DATA_BLOCK "DB_MFC_ErrorCode"
{ S7_Optimized_Access := 'TRUE' }
VERSION : 0.1
NON_RETAIN
   VAR
      PEC { ExternalAccessible := 'False'; ExternalVisible := 'False'; ExternalWritable := 'False'} : Struct
         Jam { ExternalAccessible := 'False'; ExternalVisible := 'False'; ExternalWritable := 'False'} : Int;
      END_STRUCT;
      PECUpdate { ExternalAccessible := 'False'; ExternalVisible := 'False'; ExternalWritable := 'False'} : Struct
         TooManyLost { ExternalAccessible := 'False'; ExternalVisible := 'False'; ExternalWritable := 'False'} : Int;
         LowPerformance { ExternalAccessible := 'False'; ExternalVisible := 'False'; ExternalWritable := 'False'} : Int;
         Jam { ExternalAccessible := 'False'; ExternalVisible := 'False'; ExternalWritable := 'False'} : Int;
      END_STRUCT;
      VFD { ExternalAccessible := 'False'; ExternalVisible := 'False'; ExternalWritable := 'False'} : Struct
         PNSlaveNotonline { ExternalAccessible := 'False'; ExternalVisible := 'False'; ExternalWritable := 'False'} : Int;
         PNSlaveError { ExternalAccessible := 'False'; ExternalVisible := 'False'; ExternalWritable := 'False'} : Int;
         InternalError { ExternalAccessible := 'False'; ExternalVisible := 'False'; ExternalWritable := 'False'} : Int;
         InternalWarning { ExternalAccessible := 'False'; ExternalVisible := 'False'; ExternalWritable := 'False'} : Int;
         CommunicationErrorMovikit { ExternalAccessible := 'False'; ExternalVisible := 'False'; ExternalWritable := 'False'} : Int;
         VFDRunningFeedbackError { ExternalAccessible := 'False'; ExternalVisible := 'False'; ExternalWritable := 'False'} : Int;
         PNSlaveWarning { ExternalAccessible := 'False'; ExternalVisible := 'False'; ExternalWritable := 'False'} : Int;
      END_STRUCT;
      Conveyor { ExternalAccessible := 'False'; ExternalVisible := 'False'; ExternalWritable := 'False'} : Struct
         ErrorCode { ExternalAccessible := 'False'; ExternalVisible := 'False'; ExternalWritable := 'False'} : Int;
         SubErrorCode { ExternalAccessible := 'False'; ExternalVisible := 'False'; ExternalWritable := 'False'} : Int;
         PNSlaveNotonline { ExternalAccessible := 'False'; ExternalVisible := 'False'; ExternalWritable := 'False'} : Int;
         PNSlaveError { ExternalAccessible := 'False'; ExternalVisible := 'False'; ExternalWritable := 'False'} : Int;
         InternalError { ExternalAccessible := 'False'; ExternalVisible := 'False'; ExternalWritable := 'False'} : Int;
         InternalWarning { ExternalAccessible := 'False'; ExternalVisible := 'False'; ExternalWritable := 'False'} : Int;
         CommunicationErrorMovikit { ExternalAccessible := 'False'; ExternalVisible := 'False'; ExternalWritable := 'False'} : Int;
         VFDRunningFeedbackError { ExternalAccessible := 'False'; ExternalVisible := 'False'; ExternalWritable := 'False'} : Int;
         PNSlaveWarning { ExternalAccessible := 'False'; ExternalVisible := 'False'; ExternalWritable := 'False'} : Int;
      END_STRUCT;
      Caljan { ExternalAccessible := 'False'; ExternalVisible := 'False'; ExternalWritable := 'False'} : Struct
         PNSlaveNotOnline { ExternalAccessible := 'False'; ExternalVisible := 'False'; ExternalWritable := 'False'} : Int;
         PNSlaveError { ExternalAccessible := 'False'; ExternalVisible := 'False'; ExternalWritable := 'False'} : Int;
         PNSlaveWarning { ExternalAccessible := 'False'; ExternalVisible := 'False'; ExternalWritable := 'False'} : Int;
         Disabled { ExternalAccessible := 'False'; ExternalVisible := 'False'; ExternalWritable := 'False'} : Int;
         VFDError { ExternalAccessible := 'False'; ExternalVisible := 'False'; ExternalWritable := 'False'} : Int;
         NotHealthy { ExternalAccessible := 'False'; ExternalVisible := 'False'; ExternalWritable := 'False'} : Int;
         StoreMode { ExternalAccessible := 'False'; ExternalVisible := 'False'; ExternalWritable := 'False'} : Int;
         RunMode { ExternalAccessible := 'False'; ExternalVisible := 'False'; ExternalWritable := 'False'} : Int;
         ChuteBlocked { ExternalAccessible := 'False'; ExternalVisible := 'False'; ExternalWritable := 'False'} : Int;
         Jam { ExternalAccessible := 'False'; ExternalVisible := 'False'; ExternalWritable := 'False'} : Int;
      END_STRUCT;
      ArmDiverter { ExternalAccessible := 'False'; ExternalVisible := 'False'; ExternalWritable := 'False'} : Struct
         TimeoutError { ExternalAccessible := 'False'; ExternalVisible := 'False'; ExternalWritable := 'False'} : Int;
         LimitHomeError { ExternalAccessible := 'False'; ExternalVisible := 'False'; ExternalWritable := 'False'} : Int;
         LimitDivertError { ExternalAccessible := 'False'; ExternalVisible := 'False'; ExternalWritable := 'False'} : Int;
         PXHomeError { ExternalAccessible := 'False'; ExternalVisible := 'False'; ExternalWritable := 'False'} : Int;
         PXDivertError { ExternalAccessible := 'False'; ExternalVisible := 'False'; ExternalWritable := 'False'} : Int;
         AtHomePosition { ExternalAccessible := 'False'; ExternalVisible := 'False'; ExternalWritable := 'False'} : Int;
         AtDivertPosition { ExternalAccessible := 'False'; ExternalVisible := 'False'; ExternalWritable := 'False'} : Int;
         ReferencError { ExternalAccessible := 'False'; ExternalVisible := 'False'; ExternalWritable := 'False'} : Int;
         ParcelDivertError { ExternalAccessible := 'False'; ExternalVisible := 'False'; ExternalWritable := 'False'} : Int;
      END_STRUCT;
      MCP { ExternalAccessible := 'False'; ExternalVisible := 'False'; ExternalWritable := 'False'} : Struct
         PN_PN_MSP_PNSlaveNotOnline { ExternalAccessible := 'False'; ExternalVisible := 'False'; ExternalWritable := 'False'} : Int;   // PNPN coupler is not online
         PN_PN_MSP_PNSlaveError { ExternalAccessible := 'False'; ExternalVisible := 'False'; ExternalWritable := 'False'} : Int;   // PNPN coupler has an error
         PN_PN_MSP_PNSlaveWarning { ExternalAccessible := 'False'; ExternalVisible := 'False'; ExternalWritable := 'False'} : Int;   // PNPN coupler has a warning
         IOModule_PNSlaveNotOnline { ExternalAccessible := 'False'; ExternalVisible := 'False'; ExternalWritable := 'False'} : Int;   // I/O Module is not online
         IOModule_PNSlaveError { ExternalAccessible := 'False'; ExternalVisible := 'False'; ExternalWritable := 'False'} : Int;   // I/O Module has an error
         IOModule_PNSlaveWarning { ExternalAccessible := 'False'; ExternalVisible := 'False'; ExternalWritable := 'False'} : Int;   // I/O Module has a warning
         ScalanceSwitchPNSlaveNotOnline { ExternalAccessible := 'False'; ExternalVisible := 'False'; ExternalWritable := 'False'} : Int;   // Scalance switch is not online (Switch 1)
         ScalanceSwitchPNSlaveError { ExternalAccessible := 'False'; ExternalVisible := 'False'; ExternalWritable := 'False'} : Int;   // Scalance switch has an error (Switch 1)
         ScalanceSwitchPNSlaveWarning { ExternalAccessible := 'False'; ExternalVisible := 'False'; ExternalWritable := 'False'} : Int;   // Scalance switch has a warning (Switch 1)
         "2ndScalanceSwitchPNSlaveNotOnline" { ExternalAccessible := 'False'; ExternalVisible := 'False'; ExternalWritable := 'False'} : Int;   // Scalance switch is not online (Switch 2)
         "2ndScalanceSwitchPNSlaveError" { ExternalAccessible := 'False'; ExternalVisible := 'False'; ExternalWritable := 'False'} : Int;   // Scalance switch has an error (Switch 2)
         "2ndScalanceSwitchPNSlaveWarning" { ExternalAccessible := 'False'; ExternalVisible := 'False'; ExternalWritable := 'False'} : Int;   // Scalance switch has a warning (Switch 2)
         Singulator_PNSlaveNotOnline { ExternalAccessible := 'False'; ExternalVisible := 'False'; ExternalWritable := 'False'} : Int;   // Singulator coupler is not online
         Singulator_PNSlaveError { ExternalAccessible := 'False'; ExternalVisible := 'False'; ExternalWritable := 'False'} : Int;   // Singulator coupler has an error
         Singulator_PNSlaveWarning { ExternalAccessible := 'False'; ExternalVisible := 'False'; ExternalWritable := 'False'} : Int;   // Singulator coupler has a warning
         IPS_PNSlaveNotOnline { ExternalAccessible := 'False'; ExternalVisible := 'False'; ExternalWritable := 'False'} : Int;   // IPS is not online
         IPS_PNSlaveError { ExternalAccessible := 'False'; ExternalVisible := 'False'; ExternalWritable := 'False'} : Int;   // IPS has an error
         IPS_PNSlaveWarning { ExternalAccessible := 'False'; ExternalVisible := 'False'; ExternalWritable := 'False'} : Int;   // IPS has a warning
         UPSSwitchTripped { ExternalAccessible := 'False'; ExternalVisible := 'False'; ExternalWritable := 'False'} : Int;   // Unit Power Supply switch tripped
         FireAlarmActive { ExternalAccessible := 'False'; ExternalVisible := 'False'; ExternalWritable := 'False'} : Int;   // Fire alarm active when the signal is true
         PS_201T1_Tripped { ExternalAccessible := 'False'; ExternalVisible := 'False'; ExternalWritable := 'False'} : Int;   // TRUE if power supply 201T1 tripped
         "230VAC_CB101F4Tripped" { ExternalAccessible := 'False'; ExternalVisible := 'False'; ExternalWritable := 'False'} : Int;   // TRUE if MCP circuit breaker 101F4 tripped
         "230VAC_CB102F1Tripped" { ExternalAccessible := 'False'; ExternalVisible := 'False'; ExternalWritable := 'False'} : Int;   // TRUE if MCP circuit breaker 102F1 tripped
         "24VDC_CB201F1Tripped" { ExternalAccessible := 'False'; ExternalVisible := 'False'; ExternalWritable := 'False'} : Int;   // TRUE if MCP circuit breaker 201F1 tripped
         "24VDC_CB205F5Tripped" { ExternalAccessible := 'False'; ExternalVisible := 'False'; ExternalWritable := 'False'} : Int;   // TRUE if MCP circuit breaker 205F5 tripped
         Spare_1 { ExternalAccessible := 'False'; ExternalVisible := 'False'; ExternalWritable := 'False'} : Int;   // Spare
         Spare_2 { ExternalAccessible := 'False'; ExternalVisible := 'False'; ExternalWritable := 'False'} : Int;   // Spare
         Spare_3 { ExternalAccessible := 'False'; ExternalVisible := 'False'; ExternalWritable := 'False'} : Int;   // Spare
         RackSlotError { ExternalAccessible := 'False'; ExternalVisible := 'False'; ExternalWritable := 'False'} : Array[0..31] of Int;   // One of the main rack slots has an error
         IOModuleSlotError { ExternalAccessible := 'False'; ExternalVisible := 'False'; ExternalWritable := 'False'} : Array[0..31] of Int;   // Module error
      END_STRUCT;
      RIO { ExternalAccessible := 'False'; ExternalVisible := 'False'; ExternalWritable := 'False'} : Struct
         PNSlaveNotOnline { ExternalAccessible := 'False'; ExternalVisible := 'False'; ExternalWritable := 'False'} : Int;
         PNSlaveError { ExternalAccessible := 'False'; ExternalVisible := 'False'; ExternalWritable := 'False'} : Int;
         PNSlaveWarning { ExternalAccessible := 'False'; ExternalVisible := 'False'; ExternalWritable := 'False'} : Int;
         ET200sp_ErrorModule { ExternalAccessible := 'False'; ExternalVisible := 'False'; ExternalWritable := 'False'} : Array[0..31] of Int;
      END_STRUCT;
      Connect { ExternalAccessible := 'False'; ExternalVisible := 'False'; ExternalWritable := 'False'} : Struct
         CommunicationFault { ExternalAccessible := 'False'; ExternalVisible := 'False'; ExternalWritable := 'False'} : Int;
      END_STRUCT;
      ConveyorInterface { ExternalAccessible := 'False'; ExternalVisible := 'False'; ExternalWritable := 'False'} : Struct
         InternalErrorTracking { ExternalAccessible := 'False'; ExternalVisible := 'False'; ExternalWritable := 'False'} : Int;
         InternalWarningTracking { ExternalAccessible := 'False'; ExternalVisible := 'False'; ExternalWritable := 'False'} : Int;
         Disconnected { ExternalAccessible := 'False'; ExternalVisible := 'False'; ExternalWritable := 'False'} : Int;
      END_STRUCT;
      PDP { ExternalAccessible := 'False'; ExternalVisible := 'False'; ExternalWritable := 'False'} : Struct
         CircuitBreakersTripped { ExternalAccessible := 'False'; ExternalVisible := 'False'; ExternalWritable := 'False'} : Int;
         CircuitBreakerStateF100_F200_F300 { ExternalAccessible := 'False'; ExternalVisible := 'False'; ExternalWritable := 'False'} : Int;
         CircuitBreakerStatePM { ExternalAccessible := 'False'; ExternalVisible := 'False'; ExternalWritable := 'False'} : Int;
         CircuitBreakerTrippedF101 { ExternalAccessible := 'False'; ExternalVisible := 'False'; ExternalWritable := 'False'} : Int;
         CircuitBreakerTrippedF102 { ExternalAccessible := 'False'; ExternalVisible := 'False'; ExternalWritable := 'False'} : Int;
         CircuitBreakerTrippedF103 { ExternalAccessible := 'False'; ExternalVisible := 'False'; ExternalWritable := 'False'} : Int;
         CircuitBreakerTrippedF104 { ExternalAccessible := 'False'; ExternalVisible := 'False'; ExternalWritable := 'False'} : Int;
         CircuitBreakerTrippedF105 { ExternalAccessible := 'False'; ExternalVisible := 'False'; ExternalWritable := 'False'} : Int;
         CircuitBreakerTrippedF106 { ExternalAccessible := 'False'; ExternalVisible := 'False'; ExternalWritable := 'False'} : Int;
         CircuitBreakerTrippedF107 { ExternalAccessible := 'False'; ExternalVisible := 'False'; ExternalWritable := 'False'} : Int;
         CircuitBreakerTrippedF108 { ExternalAccessible := 'False'; ExternalVisible := 'False'; ExternalWritable := 'False'} : Int;
         CircuitBreakerTrippedF109 { ExternalAccessible := 'False'; ExternalVisible := 'False'; ExternalWritable := 'False'} : Int;
         CircuitBreakerTrippedF110 { ExternalAccessible := 'False'; ExternalVisible := 'False'; ExternalWritable := 'False'} : Int;
         CircuitBreakerTrippedF111 { ExternalAccessible := 'False'; ExternalVisible := 'False'; ExternalWritable := 'False'} : Int;
         CircuitBreakerTrippedF112 { ExternalAccessible := 'False'; ExternalVisible := 'False'; ExternalWritable := 'False'} : Int;
         CircuitBreakerTrippedF113 { ExternalAccessible := 'False'; ExternalVisible := 'False'; ExternalWritable := 'False'} : Int;
         CircuitBreakerTrippedF114 { ExternalAccessible := 'False'; ExternalVisible := 'False'; ExternalWritable := 'False'} : Int;
         CircuitBreakerTrippedF115 { ExternalAccessible := 'False'; ExternalVisible := 'False'; ExternalWritable := 'False'} : Int;
         CircuitBreakerTrippedF116 { ExternalAccessible := 'False'; ExternalVisible := 'False'; ExternalWritable := 'False'} : Int;
         CircuitBreakerTrippedF117 { ExternalAccessible := 'False'; ExternalVisible := 'False'; ExternalWritable := 'False'} : Int;
         CircuitBreakerTrippedF118 { ExternalAccessible := 'False'; ExternalVisible := 'False'; ExternalWritable := 'False'} : Int;
         CircuitBreakerTrippedF119 { ExternalAccessible := 'False'; ExternalVisible := 'False'; ExternalWritable := 'False'} : Int;
         CircuitBreakerTrippedF120 { ExternalAccessible := 'False'; ExternalVisible := 'False'; ExternalWritable := 'False'} : Int;
         CircuitBreakerTrippedF121 { ExternalAccessible := 'False'; ExternalVisible := 'False'; ExternalWritable := 'False'} : Int;
         CircuitBreakerTrippedF122 { ExternalAccessible := 'False'; ExternalVisible := 'False'; ExternalWritable := 'False'} : Int;
         CircuitBreakerTrippedF123 { ExternalAccessible := 'False'; ExternalVisible := 'False'; ExternalWritable := 'False'} : Int;
         CircuitBreakerTrippedF124 { ExternalAccessible := 'False'; ExternalVisible := 'False'; ExternalWritable := 'False'} : Int;
         CircuitBreakerTrippedF125 { ExternalAccessible := 'False'; ExternalVisible := 'False'; ExternalWritable := 'False'} : Int;
         CircuitBreakerTrippedF126 { ExternalAccessible := 'False'; ExternalVisible := 'False'; ExternalWritable := 'False'} : Int;
         CircuitBreakerTrippedF127 { ExternalAccessible := 'False'; ExternalVisible := 'False'; ExternalWritable := 'False'} : Int;
         CircuitBreakerTrippedF128 { ExternalAccessible := 'False'; ExternalVisible := 'False'; ExternalWritable := 'False'} : Int;
         CircuitBreakerTrippedF129 { ExternalAccessible := 'False'; ExternalVisible := 'False'; ExternalWritable := 'False'} : Int;
         CircuitBreakerTrippedF130 { ExternalAccessible := 'False'; ExternalVisible := 'False'; ExternalWritable := 'False'} : Int;
         CircuitBreakerTrippedF131 { ExternalAccessible := 'False'; ExternalVisible := 'False'; ExternalWritable := 'False'} : Int;
         CircuitBreakerTrippedF132 { ExternalAccessible := 'False'; ExternalVisible := 'False'; ExternalWritable := 'False'} : Int;
         CircuitBreakerTrippedF133 { ExternalAccessible := 'False'; ExternalVisible := 'False'; ExternalWritable := 'False'} : Int;
         CircuitBreakerTrippedF134 { ExternalAccessible := 'False'; ExternalVisible := 'False'; ExternalWritable := 'False'} : Int;
         CircuitBreakerTrippedF135 { ExternalAccessible := 'False'; ExternalVisible := 'False'; ExternalWritable := 'False'} : Int;
         CircuitBreakerTrippedF201 { ExternalAccessible := 'False'; ExternalVisible := 'False'; ExternalWritable := 'False'} : Int;
         CircuitBreakerTrippedF202 { ExternalAccessible := 'False'; ExternalVisible := 'False'; ExternalWritable := 'False'} : Int;
         CircuitBreakerTrippedF203 { ExternalAccessible := 'False'; ExternalVisible := 'False'; ExternalWritable := 'False'} : Int;
         CircuitBreakerTrippedF204 { ExternalAccessible := 'False'; ExternalVisible := 'False'; ExternalWritable := 'False'} : Int;
         CircuitBreakerTrippedF205 { ExternalAccessible := 'False'; ExternalVisible := 'False'; ExternalWritable := 'False'} : Int;
         CircuitBreakerTrippedF206 { ExternalAccessible := 'False'; ExternalVisible := 'False'; ExternalWritable := 'False'} : Int;
         CircuitBreakerTrippedF207 { ExternalAccessible := 'False'; ExternalVisible := 'False'; ExternalWritable := 'False'} : Int;
         CircuitBreakerTrippedF208 { ExternalAccessible := 'False'; ExternalVisible := 'False'; ExternalWritable := 'False'} : Int;
         CircuitBreakerTrippedF209 { ExternalAccessible := 'False'; ExternalVisible := 'False'; ExternalWritable := 'False'} : Int;
         CircuitBreakerTrippedF210 { ExternalAccessible := 'False'; ExternalVisible := 'False'; ExternalWritable := 'False'} : Int;
         CircuitBreakerTrippedF211 { ExternalAccessible := 'False'; ExternalVisible := 'False'; ExternalWritable := 'False'} : Int;
         CircuitBreakerTrippedF212 { ExternalAccessible := 'False'; ExternalVisible := 'False'; ExternalWritable := 'False'} : Int;
         CircuitBreakerTrippedF213 { ExternalAccessible := 'False'; ExternalVisible := 'False'; ExternalWritable := 'False'} : Int;
         CircuitBreakerTrippedF214 { ExternalAccessible := 'False'; ExternalVisible := 'False'; ExternalWritable := 'False'} : Int;
         CircuitBreakerTrippedF215 { ExternalAccessible := 'False'; ExternalVisible := 'False'; ExternalWritable := 'False'} : Int;
         CircuitBreakerTrippedF216 { ExternalAccessible := 'False'; ExternalVisible := 'False'; ExternalWritable := 'False'} : Int;
         CircuitBreakerTrippedF217 { ExternalAccessible := 'False'; ExternalVisible := 'False'; ExternalWritable := 'False'} : Int;
         CircuitBreakerTrippedF218 { ExternalAccessible := 'False'; ExternalVisible := 'False'; ExternalWritable := 'False'} : Int;
         CircuitBreakerTrippedF219 { ExternalAccessible := 'False'; ExternalVisible := 'False'; ExternalWritable := 'False'} : Int;
         CircuitBreakerTrippedF220 { ExternalAccessible := 'False'; ExternalVisible := 'False'; ExternalWritable := 'False'} : Int;
         CircuitBreakerTrippedF221 { ExternalAccessible := 'False'; ExternalVisible := 'False'; ExternalWritable := 'False'} : Int;
         CircuitBreakerTrippedF222 { ExternalAccessible := 'False'; ExternalVisible := 'False'; ExternalWritable := 'False'} : Int;
         CircuitBreakerTrippedF223 { ExternalAccessible := 'False'; ExternalVisible := 'False'; ExternalWritable := 'False'} : Int;
         CircuitBreakerTrippedF224 { ExternalAccessible := 'False'; ExternalVisible := 'False'; ExternalWritable := 'False'} : Int;
         CircuitBreakerTrippedF225 { ExternalAccessible := 'False'; ExternalVisible := 'False'; ExternalWritable := 'False'} : Int;
         CircuitBreakerTrippedF226 { ExternalAccessible := 'False'; ExternalVisible := 'False'; ExternalWritable := 'False'} : Int;
         CircuitBreakerTrippedF227 { ExternalAccessible := 'False'; ExternalVisible := 'False'; ExternalWritable := 'False'} : Int;
         CircuitBreakerTrippedF228 { ExternalAccessible := 'False'; ExternalVisible := 'False'; ExternalWritable := 'False'} : Int;
         CircuitBreakerTrippedF229 { ExternalAccessible := 'False'; ExternalVisible := 'False'; ExternalWritable := 'False'} : Int;
         CircuitBreakerTrippedF501 { ExternalAccessible := 'False'; ExternalVisible := 'False'; ExternalWritable := 'False'} : Int;
         CircuitBreakerTrippedF502 { ExternalAccessible := 'False'; ExternalVisible := 'False'; ExternalWritable := 'False'} : Int;
         CircuitBreakerTrippedF503 { ExternalAccessible := 'False'; ExternalVisible := 'False'; ExternalWritable := 'False'} : Int;
         CircuitBreakerTrippedF504 { ExternalAccessible := 'False'; ExternalVisible := 'False'; ExternalWritable := 'False'} : Int;
         CircuitBreakerTrippedF505 { ExternalAccessible := 'False'; ExternalVisible := 'False'; ExternalWritable := 'False'} : Int;
         CircuitBreakerTrippedF506 { ExternalAccessible := 'False'; ExternalVisible := 'False'; ExternalWritable := 'False'} : Int;
         CircuitBreakerTrippedF507 { ExternalAccessible := 'False'; ExternalVisible := 'False'; ExternalWritable := 'False'} : Int;
         CircuitBreakerTrippedF508 { ExternalAccessible := 'False'; ExternalVisible := 'False'; ExternalWritable := 'False'} : Int;
         CircuitBreakerTrippedF509 { ExternalAccessible := 'False'; ExternalVisible := 'False'; ExternalWritable := 'False'} : Int;
         CircuitBreakerTrippedF510 { ExternalAccessible := 'False'; ExternalVisible := 'False'; ExternalWritable := 'False'} : Int;
         CircuitBreakerTrippedF511 { ExternalAccessible := 'False'; ExternalVisible := 'False'; ExternalWritable := 'False'} : Int;
         CircuitBreakerTrippedF512 { ExternalAccessible := 'False'; ExternalVisible := 'False'; ExternalWritable := 'False'} : Int;
      END_STRUCT;
      TCPIPConnection { ExternalAccessible := 'False'; ExternalVisible := 'False'; ExternalWritable := 'False'} : Struct
         CommunicationFault { ExternalAccessible := 'False'; ExternalVisible := 'False'; ExternalWritable := 'False'} : Int;
      END_STRUCT;
      PNNode { ExternalAccessible := 'False'; ExternalVisible := 'False'; ExternalWritable := 'False'} : Struct
         PNSlaveNotOnline { ExternalAccessible := 'False'; ExternalVisible := 'False'; ExternalWritable := 'False'} : Int;
         PNSlaveError { ExternalAccessible := 'False'; ExternalVisible := 'False'; ExternalWritable := 'False'} : Int;
         PNSlaveWarning { ExternalAccessible := 'False'; ExternalVisible := 'False'; ExternalWritable := 'False'} : Int;
      END_STRUCT;
      EStop { ExternalAccessible := 'False'; ExternalVisible := 'False'; ExternalWritable := 'False'} : Struct
         EStop { ExternalAccessible := 'False'; ExternalVisible := 'False'; ExternalWritable := 'False'} : Int;
      END_STRUCT;
      Outfeed2States { ExternalAccessible := 'False'; ExternalVisible := 'False'; ExternalWritable := 'False'} : Struct
         ChuteFull { ExternalAccessible := 'False'; ExternalVisible := 'False'; ExternalWritable := 'False'} : Int;
         ChuteHalfFull { ExternalAccessible := 'False'; ExternalVisible := 'False'; ExternalWritable := 'False'} : Int;
         ChuteDisabled { ExternalAccessible := 'False'; ExternalVisible := 'False'; ExternalWritable := 'False'} : Int;
      END_STRUCT;
      Rapiscan { ExternalAccessible := 'False'; ExternalVisible := 'False'; ExternalWritable := 'False'} : Struct
         XrayEnergised { ExternalAccessible := 'False'; ExternalVisible := 'False'; ExternalWritable := 'False'} : Int;
         XrayFault { ExternalAccessible := 'False'; ExternalVisible := 'False'; ExternalWritable := 'False'} : Int;
         XrayRdyRCV { ExternalAccessible := 'False'; ExternalVisible := 'False'; ExternalWritable := 'False'} : Int;
         XrayRdySend { ExternalAccessible := 'False'; ExternalVisible := 'False'; ExternalWritable := 'False'} : Int;
         BagScanning { ExternalAccessible := 'False'; ExternalVisible := 'False'; ExternalWritable := 'False'} : Int;
         TransportMode { ExternalAccessible := 'False'; ExternalVisible := 'False'; ExternalWritable := 'False'} : Int;
         BackBelt { ExternalAccessible := 'False'; ExternalVisible := 'False'; ExternalWritable := 'False'} : Int;
      END_STRUCT;
      BiDirectional { ExternalAccessible := 'False'; ExternalVisible := 'False'; ExternalWritable := 'False'} : Struct
         InfeedModeRequested { ExternalAccessible := 'False'; ExternalVisible := 'False'; ExternalWritable := 'False'} : Int;
         OutfeedModeRequested { ExternalAccessible := 'False'; ExternalVisible := 'False'; ExternalWritable := 'False'} : Int;
         InfeedModeActive { ExternalAccessible := 'False'; ExternalVisible := 'False'; ExternalWritable := 'False'} : Int;
         OutfeedModeActive { ExternalAccessible := 'False'; ExternalVisible := 'False'; ExternalWritable := 'False'} : Int;
         InfeedModeReady { ExternalAccessible := 'False'; ExternalVisible := 'False'; ExternalWritable := 'False'} : Int;
         OutfeedModeReady { ExternalAccessible := 'False'; ExternalVisible := 'False'; ExternalWritable := 'False'} : Int;
      END_STRUCT;
      DimensionsCheck_v2 { ExternalAccessible := 'False'; ExternalVisible := 'False'; ExternalWritable := 'False'} : Struct
         ParcelTooLongError { ExternalAccessible := 'False'; ExternalVisible := 'False'; ExternalWritable := 'False'} : Int;
         ParcelTooShortError { ExternalAccessible := 'False'; ExternalVisible := 'False'; ExternalWritable := 'False'} : Int;
         ParcelTooHighError { ExternalAccessible := 'False'; ExternalVisible := 'False'; ExternalWritable := 'False'} : Int;
         ParcelTooLowError { ExternalAccessible := 'False'; ExternalVisible := 'False'; ExternalWritable := 'False'} : Int;
         ParcelTooWideError { ExternalAccessible := 'False'; ExternalVisible := 'False'; ExternalWritable := 'False'} : Int;
         ParcelTooNarrowError { ExternalAccessible := 'False'; ExternalVisible := 'False'; ExternalWritable := 'False'} : Int;
         IncorrectParcelOrientationError { ExternalAccessible := 'False'; ExternalVisible := 'False'; ExternalWritable := 'False'} : Int;
         GeneralError { ExternalAccessible := 'False'; ExternalVisible := 'False'; ExternalWritable := 'False'} : Int;
         DisabledGeneralFunctionality { ExternalAccessible := 'False'; ExternalVisible := 'False'; ExternalWritable := 'False'} : Int;
         DisabledTooLongParcel { ExternalAccessible := 'False'; ExternalVisible := 'False'; ExternalWritable := 'False'} : Int;
         DisabledTooShortParcelError { ExternalAccessible := 'False'; ExternalVisible := 'False'; ExternalWritable := 'False'} : Int;
         DisabledTooHighParcelError { ExternalAccessible := 'False'; ExternalVisible := 'False'; ExternalWritable := 'False'} : Int;
         DisabledTooLowParcelError { ExternalAccessible := 'False'; ExternalVisible := 'False'; ExternalWritable := 'False'} : Int;
         DisabledTooWideParcelError { ExternalAccessible := 'False'; ExternalVisible := 'False'; ExternalWritable := 'False'} : Int;
         DisabledTooNarrowParcelError { ExternalAccessible := 'False'; ExternalVisible := 'False'; ExternalWritable := 'False'} : Int;
         DisabledParcelOrientationError { ExternalAccessible := 'False'; ExternalVisible := 'False'; ExternalWritable := 'False'} : Int;
      END_STRUCT;
      DMC { ExternalAccessible := 'False'; ExternalVisible := 'False'; ExternalWritable := 'False'} : Struct   // Old version (DMC_v1)
         ParcelTooLong { ExternalAccessible := 'False'; ExternalVisible := 'False'; ExternalWritable := 'False'} : Int;
         ParcelTooShort { ExternalAccessible := 'False'; ExternalVisible := 'False'; ExternalWritable := 'False'} : Int;
         ParcelTooHigh { ExternalAccessible := 'False'; ExternalVisible := 'False'; ExternalWritable := 'False'} : Int;
         ParcelTooLow { ExternalAccessible := 'False'; ExternalVisible := 'False'; ExternalWritable := 'False'} : Int;
         ParcelTooWide { ExternalAccessible := 'False'; ExternalVisible := 'False'; ExternalWritable := 'False'} : Int;
         ParcelTooNarrow { ExternalAccessible := 'False'; ExternalVisible := 'False'; ExternalWritable := 'False'} : Int;
         GeneralError { ExternalAccessible := 'False'; ExternalVisible := 'False'; ExternalWritable := 'False'} : Int;
         IncorrectParcelOrientationError { ExternalAccessible := 'False'; ExternalVisible := 'False'; ExternalWritable := 'False'} : Int;
         DisabledGeneralFunctionality { ExternalAccessible := 'False'; ExternalVisible := 'False'; ExternalWritable := 'False'} : Int;
         DisabledTooLongParcel { ExternalAccessible := 'False'; ExternalVisible := 'False'; ExternalWritable := 'False'} : Int;
         DisabledTooShortParcelError { ExternalAccessible := 'False'; ExternalVisible := 'False'; ExternalWritable := 'False'} : Int;
         DisabledTooHighParcelError { ExternalAccessible := 'False'; ExternalVisible := 'False'; ExternalWritable := 'False'} : Int;
         DisabledTooLowParcelError { ExternalAccessible := 'False'; ExternalVisible := 'False'; ExternalWritable := 'False'} : Int;
         DisabledTooWideParcelError { ExternalAccessible := 'False'; ExternalVisible := 'False'; ExternalWritable := 'False'} : Int;
         DisabledTooNarrowParcelError { ExternalAccessible := 'False'; ExternalVisible := 'False'; ExternalWritable := 'False'} : Int;
         DisabledParcelOrientationError { ExternalAccessible := 'False'; ExternalVisible := 'False'; ExternalWritable := 'False'} : Int;
      END_STRUCT;
      Encoder { ExternalAccessible := 'False'; ExternalVisible := 'False'; ExternalWritable := 'False'} : Struct
         InvalidValue { ExternalAccessible := 'False'; ExternalVisible := 'False'; ExternalWritable := 'False'} : Int;
         RunningFeedbackError { ExternalAccessible := 'False'; ExternalVisible := 'False'; ExternalWritable := 'False'} : Int;
      END_STRUCT;
      CPG { ExternalAccessible := 'False'; ExternalVisible := 'False'; ExternalWritable := 'False'} : Struct
         PowerSuppliesError { ExternalAccessible := 'False'; ExternalVisible := 'False'; ExternalWritable := 'False'} : Int;
      END_STRUCT;
      ColumnLift { ExternalAccessible := 'False'; ExternalVisible := 'False'; ExternalWritable := 'False'} : Struct
         ReferenceError { ExternalAccessible := 'False'; ExternalVisible := 'False'; ExternalWritable := 'False'} : Int;
         SwitchingTimerError { ExternalAccessible := 'False'; ExternalVisible := 'False'; ExternalWritable := 'False'} : Int;
         LimitSensorUpperPosition { ExternalAccessible := 'False'; ExternalVisible := 'False'; ExternalWritable := 'False'} : Int;
         LimitSensorLowerPosition { ExternalAccessible := 'False'; ExternalVisible := 'False'; ExternalWritable := 'False'} : Int;
         UpperPosition { ExternalAccessible := 'False'; ExternalVisible := 'False'; ExternalWritable := 'False'} : Int;
         LowerPosition { ExternalAccessible := 'False'; ExternalVisible := 'False'; ExternalWritable := 'False'} : Int;
         ChuteNotInPosition { ExternalAccessible := 'False'; ExternalVisible := 'False'; ExternalWritable := 'False'} : Int;
      END_STRUCT;
      ABSwitch { ExternalAccessible := 'False'; ExternalVisible := 'False'; ExternalWritable := 'False'} : Struct
         ReferenceError { ExternalAccessible := 'False'; ExternalVisible := 'False'; ExternalWritable := 'False'} : Int;
         SwitchingTimerError { ExternalAccessible := 'False'; ExternalVisible := 'False'; ExternalWritable := 'False'} : Int;
         LimitSensorUpperPosition { ExternalAccessible := 'False'; ExternalVisible := 'False'; ExternalWritable := 'False'} : Int;
         LimitSensorLowerPosition { ExternalAccessible := 'False'; ExternalVisible := 'False'; ExternalWritable := 'False'} : Int;
         UpperSwitchArea_Err { ExternalAccessible := 'False'; ExternalVisible := 'False'; ExternalWritable := 'False'} : Int;
         LowerSwitchArea_Err { ExternalAccessible := 'False'; ExternalVisible := 'False'; ExternalWritable := 'False'} : Int;
         UpperPosition { ExternalAccessible := 'False'; ExternalVisible := 'False'; ExternalWritable := 'False'} : Int;
         LowerPosition { ExternalAccessible := 'False'; ExternalVisible := 'False'; ExternalWritable := 'False'} : Int;
      END_STRUCT;
      Retractable { ExternalAccessible := 'False'; ExternalVisible := 'False'; ExternalWritable := 'False'} : Struct
         NoHomePosition { ExternalAccessible := 'False'; ExternalVisible := 'False'; ExternalWritable := 'False'} : Int;
         Errorr { ExternalAccessible := 'False'; ExternalVisible := 'False'; ExternalWritable := 'False'} : Int;
      END_STRUCT;
      CodingBeltModes { ExternalAccessible := 'False'; ExternalVisible := 'False'; ExternalWritable := 'False'} : Struct
         Infeed_LabellingMode { ExternalAccessible := 'False'; ExternalVisible := 'False'; ExternalWritable := 'False'} : Int;
         Infeed_ContinueMode { ExternalAccessible := 'False'; ExternalVisible := 'False'; ExternalWritable := 'False'} : Int;
         Infeed_BufferMode { ExternalAccessible := 'False'; ExternalVisible := 'False'; ExternalWritable := 'False'} : Int;
         Outfeed_LabellingMode { ExternalAccessible := 'False'; ExternalVisible := 'False'; ExternalWritable := 'False'} : Int;
         Outfeed_ContinueMode { ExternalAccessible := 'False'; ExternalVisible := 'False'; ExternalWritable := 'False'} : Int;
         Outfeed_BufferMode { ExternalAccessible := 'False'; ExternalVisible := 'False'; ExternalWritable := 'False'} : Int;
         GeneralError { ExternalAccessible := 'False'; ExternalVisible := 'False'; ExternalWritable := 'False'} : Int;
         ConfigurationError { ExternalAccessible := 'False'; ExternalVisible := 'False'; ExternalWritable := 'False'} : Int;
      END_STRUCT;
      EuchnerLock { ExternalAccessible := 'False'; ExternalVisible := 'False'; ExternalWritable := 'False'} : Struct
         LockFault { ExternalAccessible := 'False'; ExternalVisible := 'False'; ExternalWritable := 'False'} : Int;
         DoorClosed { ExternalAccessible := 'False'; ExternalVisible := 'False'; ExternalWritable := 'False'} : Int;
         DoorOpened { ExternalAccessible := 'False'; ExternalVisible := 'False'; ExternalWritable := 'False'} : Int;
         BoltTongueClosed { ExternalAccessible := 'False'; ExternalVisible := 'False'; ExternalWritable := 'False'} : Int;
         Safelylocked { ExternalAccessible := 'False'; ExternalVisible := 'False'; ExternalWritable := 'False'} : Int;
         SafetyLockAckReq { ExternalAccessible := 'False'; ExternalVisible := 'False'; ExternalWritable := 'False'} : Int;
         ReqMissingAccessRights { ExternalAccessible := 'False'; ExternalVisible := 'False'; ExternalWritable := 'False'} : Int;
         ResetMissingAccessRights { ExternalAccessible := 'False'; ExternalVisible := 'False'; ExternalWritable := 'False'} : Int;
         DoorOpenedWithoutReq { ExternalAccessible := 'False'; ExternalVisible := 'False'; ExternalWritable := 'False'} : Int;
      END_STRUCT;
   END_VAR


BEGIN
   PEC.Jam := 10101;
   PECUpdate.TooManyLost := 10202;
   PECUpdate.LowPerformance := 10201;
   PECUpdate.Jam := 10203;
   VFD.PNSlaveNotonline := 10006;
   VFD.PNSlaveError := 10005;
   VFD.InternalError := 10002;
   VFD.InternalWarning := 10003;
   VFD.CommunicationErrorMovikit := 10001;
   VFD.VFDRunningFeedbackError := 10004;
   VFD.PNSlaveWarning := 10007;
   Conveyor.ErrorCode := 260;
   Conveyor.SubErrorCode := 261;
   Conveyor.PNSlaveNotonline := 262;
   Conveyor.PNSlaveError := 263;
   Conveyor.InternalError := 264;
   Conveyor.InternalWarning := 265;
   Conveyor.CommunicationErrorMovikit := 266;
   Conveyor.VFDRunningFeedbackError := 267;
   Conveyor.PNSlaveWarning := 268;
   Caljan.PNSlaveNotOnline := 10602;
   Caljan.PNSlaveError := 10603;
   Caljan.PNSlaveWarning := 10604;
   Caljan.Disabled := 10605;
   Caljan.VFDError := 10606;
   Caljan.NotHealthy := 10607;
   Caljan.StoreMode := 10609;
   Caljan.RunMode := 10610;
   Caljan.ChuteBlocked := 10608;
   Caljan.Jam := 10601;
   ArmDiverter.TimeoutError := 10701;
   ArmDiverter.LimitHomeError := 10702;
   ArmDiverter.LimitDivertError := 10703;
   ArmDiverter.PXHomeError := 10704;
   ArmDiverter.PXDivertError := 10705;
   ArmDiverter.AtHomePosition := 10706;
   ArmDiverter.AtDivertPosition := 10707;
   ArmDiverter.ReferencError := 10708;
   ArmDiverter.ParcelDivertError := 10709;
   MCP.PN_PN_MSP_PNSlaveNotOnline := 1001;
   MCP.PN_PN_MSP_PNSlaveError := 1002;
   MCP.PN_PN_MSP_PNSlaveWarning := 1003;
   MCP.IOModule_PNSlaveNotOnline := 1004;
   MCP.IOModule_PNSlaveError := 1005;
   MCP.IOModule_PNSlaveWarning := 1006;
   MCP.ScalanceSwitchPNSlaveNotOnline := 1007;
   MCP.ScalanceSwitchPNSlaveError := 1008;
   MCP.ScalanceSwitchPNSlaveWarning := 1009;
   MCP."2ndScalanceSwitchPNSlaveNotOnline" := 1010;
   MCP."2ndScalanceSwitchPNSlaveError" := 1011;
   MCP."2ndScalanceSwitchPNSlaveWarning" := 1012;
   MCP.Singulator_PNSlaveNotOnline := 1013;
   MCP.Singulator_PNSlaveError := 1014;
   MCP.Singulator_PNSlaveWarning := 1015;
   MCP.IPS_PNSlaveNotOnline := 1016;
   MCP.IPS_PNSlaveError := 1017;
   MCP.IPS_PNSlaveWarning := 1018;
   MCP.UPSSwitchTripped := 1019;
   MCP.FireAlarmActive := 1020;
   MCP.PS_201T1_Tripped := 1021;
   MCP."230VAC_CB101F4Tripped" := 1022;
   MCP."230VAC_CB102F1Tripped" := 1023;
   MCP."24VDC_CB201F1Tripped" := 1024;
   MCP."24VDC_CB205F5Tripped" := 1025;
   MCP.Spare_1 := 1026;
   MCP.Spare_2 := 1027;
   MCP.Spare_3 := 1028;
   MCP.RackSlotError[0] := 1029;
   MCP.RackSlotError[1] := 1030;
   MCP.RackSlotError[2] := 1031;
   MCP.RackSlotError[3] := 1032;
   MCP.RackSlotError[4] := 1033;
   MCP.RackSlotError[5] := 1034;
   MCP.RackSlotError[6] := 1035;
   MCP.RackSlotError[7] := 1036;
   MCP.RackSlotError[8] := 1037;
   MCP.RackSlotError[9] := 1038;
   MCP.RackSlotError[10] := 1039;
   MCP.RackSlotError[11] := 1040;
   MCP.RackSlotError[12] := 1041;
   MCP.RackSlotError[13] := 1042;
   MCP.RackSlotError[14] := 1043;
   MCP.RackSlotError[15] := 1044;
   MCP.RackSlotError[16] := 1045;
   MCP.RackSlotError[17] := 1046;
   MCP.RackSlotError[18] := 1047;
   MCP.RackSlotError[19] := 1048;
   MCP.RackSlotError[20] := 1049;
   MCP.RackSlotError[21] := 1050;
   MCP.RackSlotError[22] := 1051;
   MCP.RackSlotError[23] := 1052;
   MCP.RackSlotError[24] := 1053;
   MCP.RackSlotError[25] := 1054;
   MCP.RackSlotError[26] := 1055;
   MCP.RackSlotError[27] := 1056;
   MCP.RackSlotError[28] := 1057;
   MCP.RackSlotError[29] := 1058;
   MCP.RackSlotError[30] := 1059;
   MCP.RackSlotError[31] := 1060;
   MCP.IOModuleSlotError[0] := 1061;
   MCP.IOModuleSlotError[1] := 1062;
   MCP.IOModuleSlotError[2] := 1063;
   MCP.IOModuleSlotError[3] := 1064;
   MCP.IOModuleSlotError[4] := 1065;
   MCP.IOModuleSlotError[5] := 1066;
   MCP.IOModuleSlotError[6] := 1067;
   MCP.IOModuleSlotError[7] := 1068;
   MCP.IOModuleSlotError[8] := 1069;
   MCP.IOModuleSlotError[9] := 1070;
   MCP.IOModuleSlotError[10] := 1071;
   MCP.IOModuleSlotError[11] := 1072;
   MCP.IOModuleSlotError[12] := 1073;
   MCP.IOModuleSlotError[13] := 1074;
   MCP.IOModuleSlotError[14] := 1075;
   MCP.IOModuleSlotError[15] := 1076;
   MCP.IOModuleSlotError[16] := 1077;
   MCP.IOModuleSlotError[17] := 1078;
   MCP.IOModuleSlotError[18] := 1079;
   MCP.IOModuleSlotError[19] := 1080;
   MCP.IOModuleSlotError[20] := 1081;
   MCP.IOModuleSlotError[21] := 1082;
   MCP.IOModuleSlotError[22] := 1083;
   MCP.IOModuleSlotError[23] := 1084;
   MCP.IOModuleSlotError[24] := 1085;
   MCP.IOModuleSlotError[25] := 1086;
   MCP.IOModuleSlotError[26] := 1087;
   MCP.IOModuleSlotError[27] := 1088;
   MCP.IOModuleSlotError[28] := 1089;
   MCP.IOModuleSlotError[29] := 1090;
   MCP.IOModuleSlotError[30] := 1091;
   MCP.IOModuleSlotError[31] := 1092;
   RIO.PNSlaveNotOnline := 1201;
   RIO.PNSlaveError := 1202;
   RIO.PNSlaveWarning := 1235;
   RIO.ET200sp_ErrorModule[0] := 1203;
   RIO.ET200sp_ErrorModule[1] := 1204;
   RIO.ET200sp_ErrorModule[2] := 1205;
   RIO.ET200sp_ErrorModule[3] := 1206;
   RIO.ET200sp_ErrorModule[4] := 1207;
   RIO.ET200sp_ErrorModule[5] := 1208;
   RIO.ET200sp_ErrorModule[6] := 1209;
   RIO.ET200sp_ErrorModule[7] := 1210;
   RIO.ET200sp_ErrorModule[8] := 1211;
   RIO.ET200sp_ErrorModule[9] := 1212;
   RIO.ET200sp_ErrorModule[10] := 1213;
   RIO.ET200sp_ErrorModule[11] := 1214;
   RIO.ET200sp_ErrorModule[12] := 1215;
   RIO.ET200sp_ErrorModule[13] := 1216;
   RIO.ET200sp_ErrorModule[14] := 1217;
   RIO.ET200sp_ErrorModule[15] := 1218;
   RIO.ET200sp_ErrorModule[16] := 1219;
   RIO.ET200sp_ErrorModule[17] := 1220;
   RIO.ET200sp_ErrorModule[18] := 1221;
   RIO.ET200sp_ErrorModule[19] := 1222;
   RIO.ET200sp_ErrorModule[20] := 1223;
   RIO.ET200sp_ErrorModule[21] := 1224;
   RIO.ET200sp_ErrorModule[22] := 1225;
   RIO.ET200sp_ErrorModule[23] := 1226;
   RIO.ET200sp_ErrorModule[24] := 1227;
   RIO.ET200sp_ErrorModule[25] := 1228;
   RIO.ET200sp_ErrorModule[26] := 1229;
   RIO.ET200sp_ErrorModule[27] := 1230;
   RIO.ET200sp_ErrorModule[28] := 1231;
   RIO.ET200sp_ErrorModule[29] := 1232;
   RIO.ET200sp_ErrorModule[30] := 1233;
   RIO.ET200sp_ErrorModule[31] := 1234;
   Connect.CommunicationFault := 101;
   ConveyorInterface.InternalErrorTracking := 10301;
   ConveyorInterface.InternalWarningTracking := 10302;
   ConveyorInterface.Disconnected := 10303;
   PDP.CircuitBreakersTripped := 1101;
   PDP.CircuitBreakerStateF100_F200_F300 := 1102;
   PDP.CircuitBreakerStatePM := 1103;
   PDP.CircuitBreakerTrippedF101 := 1104;
   PDP.CircuitBreakerTrippedF102 := 1105;
   PDP.CircuitBreakerTrippedF103 := 1106;
   PDP.CircuitBreakerTrippedF104 := 1107;
   PDP.CircuitBreakerTrippedF105 := 1108;
   PDP.CircuitBreakerTrippedF106 := 1109;
   PDP.CircuitBreakerTrippedF107 := 1110;
   PDP.CircuitBreakerTrippedF108 := 1111;
   PDP.CircuitBreakerTrippedF109 := 1112;
   PDP.CircuitBreakerTrippedF110 := 1113;
   PDP.CircuitBreakerTrippedF111 := 1114;
   PDP.CircuitBreakerTrippedF112 := 1115;
   PDP.CircuitBreakerTrippedF113 := 1116;
   PDP.CircuitBreakerTrippedF114 := 1117;
   PDP.CircuitBreakerTrippedF115 := 1118;
   PDP.CircuitBreakerTrippedF116 := 1119;
   PDP.CircuitBreakerTrippedF117 := 1120;
   PDP.CircuitBreakerTrippedF118 := 1121;
   PDP.CircuitBreakerTrippedF119 := 1122;
   PDP.CircuitBreakerTrippedF120 := 1123;
   PDP.CircuitBreakerTrippedF121 := 1124;
   PDP.CircuitBreakerTrippedF122 := 1125;
   PDP.CircuitBreakerTrippedF123 := 1126;
   PDP.CircuitBreakerTrippedF124 := 1127;
   PDP.CircuitBreakerTrippedF125 := 1128;
   PDP.CircuitBreakerTrippedF126 := 1129;
   PDP.CircuitBreakerTrippedF127 := 1130;
   PDP.CircuitBreakerTrippedF128 := 1131;
   PDP.CircuitBreakerTrippedF129 := 1132;
   PDP.CircuitBreakerTrippedF130 := 1133;
   PDP.CircuitBreakerTrippedF131 := 1134;
   PDP.CircuitBreakerTrippedF132 := 1135;
   PDP.CircuitBreakerTrippedF133 := 1136;
   PDP.CircuitBreakerTrippedF134 := 1137;
   PDP.CircuitBreakerTrippedF135 := 1138;
   PDP.CircuitBreakerTrippedF201 := 1139;
   PDP.CircuitBreakerTrippedF202 := 1140;
   PDP.CircuitBreakerTrippedF203 := 1141;
   PDP.CircuitBreakerTrippedF204 := 1142;
   PDP.CircuitBreakerTrippedF205 := 1143;
   PDP.CircuitBreakerTrippedF206 := 1144;
   PDP.CircuitBreakerTrippedF207 := 1145;
   PDP.CircuitBreakerTrippedF208 := 1146;
   PDP.CircuitBreakerTrippedF209 := 1147;
   PDP.CircuitBreakerTrippedF210 := 1148;
   PDP.CircuitBreakerTrippedF211 := 1149;
   PDP.CircuitBreakerTrippedF212 := 1150;
   PDP.CircuitBreakerTrippedF213 := 1151;
   PDP.CircuitBreakerTrippedF214 := 1152;
   PDP.CircuitBreakerTrippedF215 := 1153;
   PDP.CircuitBreakerTrippedF216 := 1154;
   PDP.CircuitBreakerTrippedF217 := 1155;
   PDP.CircuitBreakerTrippedF218 := 1156;
   PDP.CircuitBreakerTrippedF219 := 1157;
   PDP.CircuitBreakerTrippedF220 := 1158;
   PDP.CircuitBreakerTrippedF221 := 1159;
   PDP.CircuitBreakerTrippedF222 := 1160;
   PDP.CircuitBreakerTrippedF223 := 1161;
   PDP.CircuitBreakerTrippedF224 := 1162;
   PDP.CircuitBreakerTrippedF225 := 1163;
   PDP.CircuitBreakerTrippedF226 := 1164;
   PDP.CircuitBreakerTrippedF227 := 1165;
   PDP.CircuitBreakerTrippedF228 := 1166;
   PDP.CircuitBreakerTrippedF229 := 1167;
   PDP.CircuitBreakerTrippedF501 := 1168;
   PDP.CircuitBreakerTrippedF502 := 1169;
   PDP.CircuitBreakerTrippedF503 := 1170;
   PDP.CircuitBreakerTrippedF504 := 1171;
   PDP.CircuitBreakerTrippedF505 := 1172;
   PDP.CircuitBreakerTrippedF506 := 1173;
   PDP.CircuitBreakerTrippedF507 := 1174;
   PDP.CircuitBreakerTrippedF508 := 1175;
   PDP.CircuitBreakerTrippedF509 := 1176;
   PDP.CircuitBreakerTrippedF510 := 1177;
   PDP.CircuitBreakerTrippedF511 := 1178;
   PDP.CircuitBreakerTrippedF512 := 1179;
   TCPIPConnection.CommunicationFault := 201;
   PNNode.PNSlaveNotOnline := 1301;
   PNNode.PNSlaveError := 1302;
   PNNode.PNSlaveWarning := 1303;
   EStop.EStop := 1401;
   Outfeed2States.ChuteFull := 10401;
   Outfeed2States.ChuteHalfFull := 10402;
   Outfeed2States.ChuteDisabled := 10403;
   Rapiscan.XrayEnergised := 11101;
   Rapiscan.XrayFault := 11102;
   Rapiscan.XrayRdyRCV := 11103;
   Rapiscan.XrayRdySend := 11104;
   Rapiscan.BagScanning := 11105;
   Rapiscan.TransportMode := 11106;
   Rapiscan.BackBelt := 11107;
   BiDirectional.InfeedModeRequested := 1601;
   BiDirectional.OutfeedModeRequested := 1602;
   BiDirectional.InfeedModeActive := 1603;
   BiDirectional.OutfeedModeActive := 1604;
   BiDirectional.InfeedModeReady := 1605;
   BiDirectional.OutfeedModeReady := 1606;
   DimensionsCheck_v2.ParcelTooLongError := 10501;
   DimensionsCheck_v2.ParcelTooShortError := 10505;
   DimensionsCheck_v2.ParcelTooHighError := 10502;
   DimensionsCheck_v2.ParcelTooLowError := 10504;
   DimensionsCheck_v2.ParcelTooWideError := 10503;
   DimensionsCheck_v2.ParcelTooNarrowError := 10506;
   DimensionsCheck_v2.IncorrectParcelOrientationError := 10508;
   DimensionsCheck_v2.GeneralError := 10507;
   DimensionsCheck_v2.DisabledGeneralFunctionality := 10509;
   DimensionsCheck_v2.DisabledTooLongParcel := 10510;
   DimensionsCheck_v2.DisabledTooShortParcelError := 10511;
   DimensionsCheck_v2.DisabledTooHighParcelError := 10512;
   DimensionsCheck_v2.DisabledTooLowParcelError := 10513;
   DimensionsCheck_v2.DisabledTooWideParcelError := 10514;
   DimensionsCheck_v2.DisabledTooNarrowParcelError := 10515;
   DimensionsCheck_v2.DisabledParcelOrientationError := 10516;
   DMC.ParcelTooLong := 10501;
   DMC.ParcelTooShort := 10505;
   DMC.ParcelTooHigh := 10502;
   DMC.ParcelTooLow := 10504;
   DMC.ParcelTooWide := 10503;
   DMC.ParcelTooNarrow := 10506;
   DMC.GeneralError := 10507;
   DMC.IncorrectParcelOrientationError := 10508;
   DMC.DisabledGeneralFunctionality := 10509;
   DMC.DisabledTooLongParcel := 10510;
   DMC.DisabledTooShortParcelError := 10511;
   DMC.DisabledTooHighParcelError := 10512;
   DMC.DisabledTooLowParcelError := 10513;
   DMC.DisabledTooWideParcelError := 10514;
   DMC.DisabledTooNarrowParcelError := 10515;
   DMC.DisabledParcelOrientationError := 10516;
   Encoder.InvalidValue := 10801;
   Encoder.RunningFeedbackError := 10802;
   CPG.PowerSuppliesError := 1501;
   ColumnLift.ReferenceError := 10901;
   ColumnLift.SwitchingTimerError := 10902;
   ColumnLift.LimitSensorUpperPosition := 10903;
   ColumnLift.LimitSensorLowerPosition := 10904;
   ColumnLift.UpperPosition := 10905;
   ColumnLift.LowerPosition := 10906;
   ColumnLift.ChuteNotInPosition := 10907;
   ABSwitch.ReferenceError := 11001;
   ABSwitch.SwitchingTimerError := 11002;
   ABSwitch.LimitSensorUpperPosition := 11003;
   ABSwitch.LimitSensorLowerPosition := 11004;
   ABSwitch.UpperSwitchArea_Err := 11005;
   ABSwitch.LowerSwitchArea_Err := 11006;
   ABSwitch.UpperPosition := 11007;
   ABSwitch.LowerPosition := 11008;
   Retractable.NoHomePosition := 11301;
   Retractable.Errorr := 11302;
   CodingBeltModes.Infeed_LabellingMode := 11201;
   CodingBeltModes.Infeed_ContinueMode := 11202;
   CodingBeltModes.Infeed_BufferMode := 11203;
   CodingBeltModes.Outfeed_LabellingMode := 11204;
   CodingBeltModes.Outfeed_ContinueMode := 11205;
   CodingBeltModes.Outfeed_BufferMode := 11206;
   CodingBeltModes.GeneralError := 11207;
   CodingBeltModes.ConfigurationError := 11208;
   EuchnerLock.LockFault := 11401;
   EuchnerLock.DoorClosed := 11402;
   EuchnerLock.DoorOpened := 11403;
   EuchnerLock.BoltTongueClosed := 11404;
   EuchnerLock.Safelylocked := 11405;
   EuchnerLock.SafetyLockAckReq := 11406;
   EuchnerLock.ReqMissingAccessRights := 11407;
   EuchnerLock.ResetMissingAccessRights := 11408;
   EuchnerLock.DoorOpenedWithoutReq := 11409;

END_DATA_BLOCK

TYPE "UDT_PDPStatus"
VERSION : 0.1
   STRUCT
      Status : Int;   // Status number
      Specific : Struct   // Specific
         CircuitBreakersTripped : Bool;   // Circuit breakers tripped when the value is true
         CircuitBreakerStateF100_F200_F300 : Bool;   // Circuit Breaker State Ok if the signal is true
         CircuitBreakerStatePM : Bool;   // Circuit Breaker State Ok if the signal is true
         CircuitBreakerTrippedF101 : Bool;   // Circuit breaker is tripped when the value is true
         CircuitBreakerTrippedF102 : Bool;   // Circuit breaker is tripped when the value is true
         CircuitBreakerTrippedF103 : Bool;   // Circuit breaker is tripped when the value is true
         CircuitBreakerTrippedF104 : Bool;   // Circuit breaker is tripped when the value is true
         CircuitBreakerTrippedF105 : Bool;   // Circuit breaker is tripped when the value is true
         CircuitBreakerTrippedF106 : Bool;   // Circuit breaker is tripped when the value is true
         CircuitBreakerTrippedF107 : Bool;   // Circuit breaker is tripped when the value is true
         CircuitBreakerTrippedF108 : Bool;   // Circuit breaker is tripped when the value is true
         CircuitBreakerTrippedF109 : Bool;   // Circuit breaker is tripped when the value is true
         CircuitBreakerTrippedF110 : Bool;   // Circuit breaker is tripped when the value is true
         CircuitBreakerTrippedF111 : Bool;   // Circuit breaker is tripped when the value is true
         CircuitBreakerTrippedF112 : Bool;   // Circuit breaker is tripped when the value is true
         CircuitBreakerTrippedF113 : Bool;   // Circuit breaker is tripped when the value is true
         CircuitBreakerTrippedF114 : Bool;   // Circuit breaker is tripped when the value is true
         CircuitBreakerTrippedF115 : Bool;   // Circuit breaker is tripped when the value is true
         CircuitBreakerTrippedF116 : Bool;   // Circuit breaker is tripped when the value is true
         CircuitBreakerTrippedF117 : Bool;   // Circuit breaker is tripped when the value is true
         CircuitBreakerTrippedF118 : Bool;   // Circuit breaker is tripped when the value is true
         CircuitBreakerTrippedF119 : Bool;   // Circuit breaker is tripped when the value is true
         CircuitBreakerTrippedF120 : Bool;   // Circuit breaker is tripped when the value is true
         CircuitBreakerTrippedF121 : Bool;   // Circuit breaker is tripped when the value is true
         CircuitBreakerTrippedF122 : Bool;   // Circuit breaker is tripped when the value is true
         CircuitBreakerTrippedF123 : Bool;   // Circuit breaker is tripped when the value is true
         CircuitBreakerTrippedF124 : Bool;   // Circuit breaker is tripped when the value is true
         CircuitBreakerTrippedF125 : Bool;   // Circuit breaker is tripped when the value is true
         CircuitBreakerTrippedF126 : Bool;   // Circuit breaker is tripped when the value is true
         CircuitBreakerTrippedF127 : Bool;   // Circuit breaker is tripped when the value is true
         CircuitBreakerTrippedF128 : Bool;   // Circuit breaker is tripped when the value is true
         CircuitBreakerTrippedF129 : Bool;   // Circuit breaker is tripped when the value is true
         CircuitBreakerTrippedF130 : Bool;   // Circuit breaker is tripped when the value is true
         CircuitBreakerTrippedF131 : Bool;   // Circuit breaker is tripped when the value is true
         CircuitBreakerTrippedF132 : Bool;   // Circuit breaker is tripped when the value is true
         CircuitBreakerTrippedF133 : Bool;   // Circuit breaker is tripped when the value is true
         CircuitBreakerTrippedF134 : Bool;   // Circuit breaker is tripped when the value is true
         CircuitBreakerTrippedF135 : Bool;   // Circuit breaker is tripped when the value is true
         CircuitBreakerTrippedF201 : Bool;   // Circuit breaker is tripped when the value is true
         CircuitBreakerTrippedF202 : Bool;   // Circuit breaker is tripped when the value is true
         CircuitBreakerTrippedF203 : Bool;   // Circuit breaker is tripped when the value is true
         CircuitBreakerTrippedF204 : Bool;   // Circuit breaker is tripped when the value is true
         CircuitBreakerTrippedF205 : Bool;   // Circuit breaker is tripped when the value is true
         CircuitBreakerTrippedF206 : Bool;   // Circuit breaker is tripped when the value is true
         CircuitBreakerTrippedF207 : Bool;   // Circuit breaker is tripped when the value is true
         CircuitBreakerTrippedF208 : Bool;   // Circuit breaker is tripped when the value is true
         CircuitBreakerTrippedF209 : Bool;   // Circuit breaker is tripped when the value is true
         CircuitBreakerTrippedF210 : Bool;   // Circuit breaker is tripped when the value is true
         CircuitBreakerTrippedF211 : Bool;   // Circuit breaker is tripped when the value is true
         CircuitBreakerTrippedF212 : Bool;   // Circuit breaker is tripped when the value is true
         CircuitBreakerTrippedF213 : Bool;   // Circuit breaker is tripped when the value is true
         CircuitBreakerTrippedF214 : Bool;   // Circuit breaker is tripped when the value is true
         CircuitBreakerTrippedF215 : Bool;   // Circuit breaker is tripped when the value is true
         CircuitBreakerTrippedF216 : Bool;   // Circuit breaker is tripped when the value is true
         CircuitBreakerTrippedF217 : Bool;   // Circuit breaker is tripped when the value is true
         CircuitBreakerTrippedF218 : Bool;   // Circuit breaker is tripped when the value is true
         CircuitBreakerTrippedF219 : Bool;   // Circuit breaker is tripped when the value is true
         CircuitBreakerTrippedF220 : Bool;   // Circuit breaker is tripped when the value is true
         CircuitBreakerTrippedF221 : Bool;   // Circuit breaker is tripped when the value is true
         CircuitBreakerTrippedF222 : Bool;   // Circuit breaker is tripped when the value is true
         CircuitBreakerTrippedF223 : Bool;   // Circuit breaker is tripped when the value is true
         CircuitBreakerTrippedF224 : Bool;   // Circuit breaker is tripped when the value is true
         CircuitBreakerTrippedF225 : Bool;   // Circuit breaker is tripped when the value is true
         CircuitBreakerTrippedF226 : Bool;   // Circuit breaker is tripped when the value is true
         CircuitBreakerTrippedF227 : Bool;   // Circuit breaker is tripped when the value is true
         CircuitBreakerTrippedF228 : Bool;   // Circuit breaker is tripped when the value is true
         CircuitBreakerTrippedF229 : Bool;   // Circuit breaker is tripped when the value is true
         CircuitBreakerTrippedF501 : Bool;   // Circuit breaker is tripped when the value is true
         CircuitBreakerTrippedF502 : Bool;   // Circuit breaker is tripped when the value is true
         CircuitBreakerTrippedF503 : Bool;   // Circuit breaker is tripped when the value is true
         CircuitBreakerTrippedF504 : Bool;   // Circuit breaker is tripped when the value is true
         CircuitBreakerTrippedF505 : Bool;   // Circuit breaker is tripped when the value is true
         CircuitBreakerTrippedF506 : Bool;   // Circuit breaker is tripped when the value is true
         CircuitBreakerTrippedF507 : Bool;   // Circuit breaker is tripped when the value is true
         CircuitBreakerTrippedF508 : Bool;   // Circuit breaker is tripped when the value is true
         CircuitBreakerTrippedF509 : Bool;   // Circuit breaker is tripped when the value is true
         CircuitBreakerTrippedF510 : Bool;   // Circuit breaker is tripped when the value is true
         CircuitBreakerTrippedF511 : Bool;   // Circuit breaker is tripped when the value is true
         CircuitBreakerTrippedF512 : Bool;   // Circuit breaker is tripped when the value is true
      END_STRUCT;
   END_STRUCT;

END_TYPE

TYPE "UDT_PNNodeStatus"
VERSION : 0.1
   STRUCT
      Status : Int;   // Status number
      Specific : Struct   // Specific structure
         PNSlaveNotOnline { ExternalAccessible := 'False'; ExternalVisible := 'False'; ExternalWritable := 'False'} : Bool;   // Profinet slave is not online
         PNSlaveError { ExternalAccessible := 'False'; ExternalVisible := 'False'; ExternalWritable := 'False'} : Bool;   // Profinet slave is in error
         PNSlaveWarning { ExternalAccessible := 'False'; ExternalVisible := 'False'; ExternalWritable := 'False'} : Bool;   // Profinet slave has  a warning
      END_STRUCT;
   END_STRUCT;

END_TYPE

FUNCTION_BLOCK "FB_TIDLost"
{ S7_Optimized_Access := 'TRUE' }
VERSION : 0.1
// ATTRIBUTES
// AUTO_NUMBER = True
// BLOCK_NUMBER = 164
// END_ATTRIBUTES
   VAR_INPUT
      i_UDT_EquipmentNumber { ExternalAccessible := 'False'; ExternalVisible := 'False'; ExternalWritable := 'False'} : "UDT_EquipmentNumber";   // Item number
      idi_TID { ExternalAccessible := 'False'; ExternalVisible := 'False'; ExternalWritable := 'False'} : DInt;   // Transport ID
      is_Reason { ExternalAccessible := 'False'; ExternalVisible := 'False'; ExternalWritable := 'False'} : Struct   // TID lost reason
         Unknown { ExternalAccessible := 'False'; ExternalVisible := 'False'; ExternalWritable := 'False'} : Bool;   // Unknown
         TIDLost { ExternalAccessible := 'False'; ExternalVisible := 'False'; ExternalWritable := 'False'} : Bool;   // TID lost
         EndOfLine { ExternalAccessible := 'False'; ExternalVisible := 'False'; ExternalWritable := 'False'} : Bool;   // End of line
         ParcelDidntArrive { ExternalAccessible := 'False'; ExternalVisible := 'False'; ExternalWritable := 'False'} : Bool;   // Parcel didn't arrave on PEC when expected
         UserDelete { ExternalAccessible := 'False'; ExternalVisible := 'False'; ExternalWritable := 'False'} : Bool;   // User delete
      END_STRUCT;
      ii_MessageGroup { ExternalAccessible := 'False'; ExternalVisible := 'False'; ExternalWritable := 'False'} : Int;   // Message group
      ix_FlagRetry { ExternalAccessible := 'False'; ExternalVisible := 'False'; ExternalWritable := 'False'} : Bool;   // TRUE when message is sent again
      idi_TimeSpan { ExternalAccessible := 'False'; ExternalVisible := 'False'; ExternalWritable := 'False'} : DInt;   // Time difference between messages
   END_VAR

   VAR_OUTPUT
      qx_Error { ExternalAccessible := 'False'; ExternalVisible := 'False'; ExternalWritable := 'False'} : Bool;   // TRUE when collective block error occurred
      qx_Warning { ExternalAccessible := 'False'; ExternalVisible := 'False'; ExternalWritable := 'False'} : Bool;   // TRUE when collective block warning occurred
   END_VAR

   VAR_IN_OUT
      iq_UDT_FifoHeader : "UDT_FifoHeader";   // FIFO header
      iqs_FifoData : Array[*] of "UDT_MessageV2";   // FIFO data
      iqdi_MessageSequenceNumber { ExternalAccessible := 'False'; ExternalVisible := 'False'; ExternalWritable := 'False'} : DInt;   // Sequence number
   END_VAR

   VAR
      ss_Status { ExternalAccessible := 'False'; ExternalVisible := 'False'; ExternalWritable := 'False'} : Struct   // Status structure
         FIFOStatus { ExternalAccessible := 'False'; ExternalVisible := 'False'; ExternalWritable := 'False'} : "UDT_FifoStatus";   // FIFO status structure
         FIFOError { ExternalAccessible := 'False'; ExternalVisible := 'False'; ExternalWritable := 'False'; S7_SetPoint := 'True'} : Bool;   // FIFO error
         FIFOWarning { ExternalAccessible := 'False'; ExternalVisible := 'False'; ExternalWritable := 'False'; S7_SetPoint := 'True'} : Bool;   // FIFO warning
         InvalidMessageArraySize { ExternalAccessible := 'False'; ExternalVisible := 'False'; ExternalWritable := 'False'} : Bool;   // Invalid message array size
         InvalidReason { ExternalAccessible := 'False'; ExternalVisible := 'False'; ExternalWritable := 'False'} : Bool;   // Invalid reason value
      END_STRUCT;
      s_UDT_MessageArray { ExternalAccessible := 'False'; ExternalVisible := 'False'; ExternalWritable := 'False'; S7_SetPoint := 'False'} : "UDT_MessageV2";   // Message byte array
      s_UDT_MessageHeader { ExternalAccessible := 'False'; ExternalVisible := 'False'; ExternalWritable := 'False'; S7_SetPoint := 'False'} : "UDT_MessageHeaderV2";   // Message header
      s_UDT_MessageBody { ExternalAccessible := 'False'; ExternalVisible := 'False'; ExternalWritable := 'False'; S7_SetPoint := 'False'} : "UDT_TIDLostBody";   // Message body
      sdi_SerializePosition { ExternalAccessible := 'False'; ExternalVisible := 'False'; ExternalWritable := 'False'} : DInt;   // Serialize position
      si_HeaderSerializeStatus { ExternalAccessible := 'False'; ExternalVisible := 'False'; ExternalWritable := 'False'} : Int;   // Header serialize status
      si_BodySerializeStatus { ExternalAccessible := 'False'; ExternalVisible := 'False'; ExternalWritable := 'False'} : Int;   // Body serialize status
      si_MaximumMessageLength { ExternalAccessible := 'False'; ExternalVisible := 'False'; ExternalWritable := 'False'} : Int;   // Maximum message length
   END_VAR

   VAR CONSTANT
      ci_BodyLength : Int := 12;   // Body length
      ci_MessageID : Int := 1478;   // Message ID
      ci_MessageLength : Int := 30;   // Message length
   END_VAR


BEGIN
	(*
	----------------------------------------------------------------------------------------
	|                                                                                      |
	|  Copyright  2023             FORTNA Europe BV                                        |
	|  All Rights Reserved         Netherlands                                             |
	|                                                                                      |
	----------------------------------------------------------------------------------------
	Version history:
	Date        | Version   | Author       | Remark
	----------------------------------------------------------------------------------------
	21/12/2022  | 1.0       | S. Nikodem   | Release TIA 17 | DHL Munich 2023
	13/03/2023  | 1.1       | S. Nieswiec  | Updated for new Baseline
	*)

	REGION 1 - FIFO header status update

	    // Mode 'S' - FIFO register status update.
	    "FC_Fifo"(ic_Mode := 'S',
	              qUDT_Status => #ss_Status.FIFOStatus,
	              qx_Error => #ss_Status.FIFOError,
	              qx_Warning => #ss_Status.FIFOWarning,
	              iqv_Data := #s_UDT_MessageArray,
	              iqUDT_FifoHeader := #iq_UDT_FifoHeader,
	              iqv_DataBuffer := #iqs_FifoData);

	END_REGION

	REGION 2 - Reason validation

	    // Unknown.
	    IF #is_Reason.Unknown
	    THEN
	        #s_UDT_MessageBody.Reason := 0;
	        #ss_Status.InvalidReason := FALSE;
	        // TID lost.
	    ELSIF #is_Reason.TIDLost
	    THEN
	        #s_UDT_MessageBody.Reason := 10;
	        #ss_Status.InvalidReason := FALSE;
	        // End of line.
	    ELSIF #is_Reason.EndOfLine
	    THEN
	        #s_UDT_MessageBody.Reason := 20;
	        #ss_Status.InvalidReason := FALSE;
	        //Parcel didn't arrive on PEC when expected
	    ELSIF #is_Reason.ParcelDidntArrive
	    THEN
	        #s_UDT_MessageBody.Reason := 30;
	        #ss_Status.InvalidReason := FALSE;
	        // User delete.
	    ELSIF #is_Reason.UserDelete
	    THEN
	        #s_UDT_MessageBody.Reason := 1000;
	        #ss_Status.InvalidReason := FALSE;
	        // There is no reason.
	    ELSE
	        #ss_Status.InvalidReason := TRUE;
	    END_IF;

	END_REGION

	REGION 3 - Message array size validation

	    // Get size of the array.
	    #si_MaximumMessageLength := "FC_GetNrOfArrayEl"(iv_Array := #s_UDT_MessageArray.Bytes);

	    // Message array size validation.
	    #ss_Status.InvalidMessageArraySize := #ci_MessageLength > #si_MaximumMessageLength;

	END_REGION

	REGION 4 - Message preparation

	    // Errors check.
	    IF NOT #ss_Status.FIFOError
	        AND NOT #ss_Status.InvalidMessageArraySize
	        AND NOT #ss_Status.InvalidReason
	    THEN
	        // FIFO full check.
	        IF NOT #iq_UDT_FifoHeader.Status.Full
	        THEN

	            REGION 4.1 - Header preparation

	                // Check sequence number. If it is equal or greater than 30000 reset it to 1.
	                IF #iqdi_MessageSequenceNumber < 30000
	                THEN
	                    #iqdi_MessageSequenceNumber += 1;
	                ELSE
	                    #iqdi_MessageSequenceNumber := 1;
	                END_IF;

	                // Write parts of the header into structure.
	                #s_UDT_MessageHeader.BodyLength := #ci_BodyLength;
	                #s_UDT_MessageHeader.FlagRetry.%X0 := #ix_FlagRetry;
	                #s_UDT_MessageHeader.Group := #ii_MessageGroup;
	                #s_UDT_MessageHeader.MessageID := #ci_MessageID;
	                #s_UDT_MessageHeader.SequenceNumber := #iqdi_MessageSequenceNumber;
	                #s_UDT_MessageHeader.TimeSpan := #idi_TimeSpan;

	                // Calculate the header checksum.
	                "FC_Checksum"(i_UDT_MessageHeader := #s_UDT_MessageHeader,
	                              qb_Checksum => #s_UDT_MessageHeader.Checksum);

	            END_REGION

	            REGION 4.2 - Convert header into array of bytes

	                // Initialize the header serialize position and convert header structure into array of bytes.
	                #sdi_SerializePosition := 0;
	                #si_HeaderSerializeStatus := Serialize(SRC_VARIABLE := #s_UDT_MessageHeader,
	                                                       DEST_ARRAY => #s_UDT_MessageArray.Bytes,
	                                                       POS := #sdi_SerializePosition);

	            END_REGION

	            REGION 4.3 - Body preparation

	                // Write parts of the message body into the structure.
	                #s_UDT_MessageBody.Group := #i_UDT_EquipmentNumber.Group;
	                #s_UDT_MessageBody.Node := #i_UDT_EquipmentNumber.Node;
	                #s_UDT_MessageBody.TLLNumber := 0;
	                #s_UDT_MessageBody.TID := #idi_TID;

	            END_REGION

	            REGION 4.4 - Convert body into array of bytes

	                // Convert message body structure into array of bytes.
	                #si_BodySerializeStatus := Serialize(SRC_VARIABLE := #s_UDT_MessageBody,
	                                                     DEST_ARRAY => #s_UDT_MessageArray.Bytes,
	                                                     POS := #sdi_SerializePosition);

	            END_REGION

	            REGION 4.5 - Write message into the FIFO buffer

	                // Mode 'W' - Write FIFO record.
	                "FC_Fifo"(ic_Mode := 'W',
	                          qUDT_Status => #ss_Status.FIFOStatus,
	                          qx_Error => #ss_Status.FIFOError,
	                          qx_Warning => #ss_Status.FIFOWarning,
	                          iqv_Data := #s_UDT_MessageArray,
	                          iqUDT_FifoHeader := #iq_UDT_FifoHeader,
	                          iqv_DataBuffer := #iqs_FifoData);

	            END_REGION

	        ELSE
	            // If FIFO is full set FIFO main and FIFO full errors.
	            #ss_Status.FIFOError := TRUE;
	            #ss_Status.FIFOStatus.FifoFull := TRUE;
	        END_IF;
	    END_IF;

	END_REGION

	REGION 5 - Status

	    // Parametrization collective error output.
	    #qx_Error :=
	    #ss_Status.InvalidMessageArraySize
	    OR #ss_Status.FIFOError
	    OR #ss_Status.InvalidReason;

	    // Parametrization collective warning output.
	    #qx_Warning := #ss_Status.FIFOWarning;

	END_REGION
END_FUNCTION_BLOCK

FUNCTION_BLOCK "FB_MFC_Visu_TCPIPReceive"
TITLE = FB_TCPIPReceive
{ S7_Optimized_Access := 'TRUE' }
AUTHOR : MHSE
FAMILY : Communication
VERSION : 2.0
// ATTRIBUTES
// AUTO_NUMBER = True
// BLOCK_NUMBER = 161
// END_ATTRIBUTES
//Function block to receive data from TCPIP.
   VAR_INPUT
      i_UDT_Connection { ExternalAccessible := 'False'; ExternalVisible := 'False'; ExternalWritable := 'False'} : "UDT_Connection";   // Connection parameters
      ix_EnableReceive { ExternalAccessible := 'False'; ExternalVisible := 'False'; ExternalWritable := 'False'} : Bool;   // TRUE when receive enable
      ii_HeaderLength { ExternalAccessible := 'False'; ExternalVisible := 'False'; ExternalWritable := 'False'} : Int;   // Message header length
      ii_BodyLengthPosition { ExternalAccessible := 'False'; ExternalVisible := 'False'; ExternalWritable := 'False'} : Int;   // Position in header where message body length value starts
   END_VAR

   VAR_OUTPUT
      qx_Error { ExternalAccessible := 'False'; ExternalVisible := 'False'; ExternalWritable := 'False'} : Bool;   // TRUE when collective block error occurred
      qx_Warning { ExternalAccessible := 'False'; ExternalVisible := 'False'; ExternalWritable := 'False'} : Bool;   // TRUE when collective block warning occurred
   END_VAR

   VAR_IN_OUT
      iq_UDT_FifoHeader : "UDT_FifoHeader";   // Fifo header
      iqs_FifoData : Variant;   // Fifo data
      iq_UDT_Statistics : "UDT_TCPIPReceiveStatistics";   // Statistic structure
   END_VAR

   VAR
      s_FB_TRCV {InstructionName := 'TRCV'; LibVersion := '4.0'; ExternalAccessible := 'False'; ExternalVisible := 'False'; ExternalWritable := 'False'; S7_SetPoint := 'False'} : TRCV;   // Siemens "TRCV" block - to receive the data from TCPIP socket
      ss_TRCV { ExternalAccessible := 'False'; ExternalVisible := 'False'; ExternalWritable := 'False'} : Struct   // TRCV block interface structure
         Enable { ExternalAccessible := 'False'; ExternalVisible := 'False'; ExternalWritable := 'False'} : Bool;   //     TRCV - Enable
         NDR { ExternalAccessible := 'False'; ExternalVisible := 'False'; ExternalWritable := 'False'} : Bool;   //     TRCV - New data available
         Busy { ExternalAccessible := 'False'; ExternalVisible := 'False'; ExternalWritable := 'False'} : Bool;   //     TRCV - Busy
         Error { ExternalAccessible := 'False'; ExternalVisible := 'False'; ExternalWritable := 'False'} : Bool;   //     TRCV - Error
         Status { ExternalAccessible := 'False'; ExternalVisible := 'False'; ExternalWritable := 'False'} : Word;   //     TRCV - Status
         ReceivedLength { ExternalAccessible := 'False'; ExternalVisible := 'False'; ExternalWritable := 'False'} : UDInt;   //     TRCV - Received length
         Data { ExternalAccessible := 'False'; ExternalVisible := 'False'; ExternalWritable := 'False'} : Array[0..120] of Byte;   //     TRCV - Data
      END_STRUCT;
      s_UDT_MessageArray { ExternalAccessible := 'False'; ExternalVisible := 'False'; ExternalWritable := 'False'; S7_SetPoint := 'False'} : "UDT_MessageV2";   // Message byte array
      s_UDT_MessagePartArray { ExternalAccessible := 'False'; ExternalVisible := 'False'; ExternalWritable := 'False'; S7_SetPoint := 'False'} : "UDT_MessageV2";   // Part of the message byte array
      ss_Status { ExternalAccessible := 'False'; ExternalVisible := 'False'; ExternalWritable := 'False'} : Struct   // Status structure
         ErrorCode { ExternalAccessible := 'False'; ExternalVisible := 'False'; ExternalWritable := 'False'} : Struct   //    Error code structure
            TRCV { ExternalAccessible := 'False'; ExternalVisible := 'False'; ExternalWritable := 'False'} : Word;   //    Siemens TRCV error code - Check documentation
         END_STRUCT;
         FIFOReceiveStatus { ExternalAccessible := 'False'; ExternalVisible := 'False'; ExternalWritable := 'False'} : "UDT_FifoStatus";   //    Receive FIFO status structure
         FIFOReceiveError { ExternalAccessible := 'False'; ExternalVisible := 'False'; ExternalWritable := 'False'; S7_SetPoint := 'True'} : Bool;   //    Receive FIFO error
         FIFOReceiveWarning { ExternalAccessible := 'False'; ExternalVisible := 'False'; ExternalWritable := 'False'; S7_SetPoint := 'True'} : Bool;   //    Receive  FIFO warning
         ReceiveError { ExternalAccessible := 'False'; ExternalVisible := 'False'; ExternalWritable := 'False'} : Bool;   //    TRCV block operation error - Check TRCVStatus
      END_STRUCT;
      sui_ReceivedMessagesOffset { ExternalAccessible := 'False'; ExternalVisible := 'False'; ExternalWritable := 'False'} : Int;   // Received message offset
      sui_ReceivedMessageLength { ExternalAccessible := 'False'; ExternalVisible := 'False'; ExternalWritable := 'False'} : UInt;   // Received message length
      sui_NumberOfReceivedMessages { ExternalAccessible := 'False'; ExternalVisible := 'False'; ExternalWritable := 'False'} : UInt;   // Number of received messages in one frame
      sui_ReceivedMessagePartLength { ExternalAccessible := 'False'; ExternalVisible := 'False'; ExternalWritable := 'False'} : UInt;   // Length of the part of received message
      si_MaximumMessageLength { ExternalAccessible := 'False'; ExternalVisible := 'False'; ExternalWritable := 'False'} : Int;   // Maximum message length
      sx_ReceivedMessagePart { ExternalAccessible := 'False'; ExternalVisible := 'False'; ExternalWritable := 'False'} : Bool;   // Received part of the message
      sx_STXFound { ExternalAccessible := 'False'; ExternalVisible := 'False'; ExternalWritable := 'False'} : Bool;   // STX in message is found
      sw_BodyLength { ExternalAccessible := 'False'; ExternalVisible := 'False'; ExternalWritable := 'False'} : Word;   // Message body length
      si_BodyLength { ExternalAccessible := 'False'; ExternalVisible := 'False'; ExternalWritable := 'False'} : Int;   // Message body length
      si_BodyLengthFirstPart { ExternalAccessible := 'False'; ExternalVisible := 'False'; ExternalWritable := 'False'} : Int;   // First part of the message body length
      si_BodyLengthSecondPart { ExternalAccessible := 'False'; ExternalVisible := 'False'; ExternalWritable := 'False'} : Int;   // Second part of the message body length
      sx_STXFoundEnd { ExternalAccessible := 'False'; ExternalVisible := 'False'; ExternalWritable := 'False'} : Bool;   // STX found on the end of first message buffer
   END_VAR

   VAR_TEMP
      ti_LC_MessageChars : Int;   //  Message chars loop counter
   END_VAR

   VAR CONSTANT
      cb_STX : Byte := 16#02;   // Start of the message sign
      cb_NULL : Byte := 16#00;   // NULL sign
   END_VAR


BEGIN
	(*
	----------------------------------------------------------------------------------------
	|                                                                                      |
	|  Copyright  2019             MHS                                                     |
	|  All Rights Reserved         Larenweg 90                                             |
	|                              5234 KC 's-Hertogenbosch,                               |
	|                              Netherlands                                             |
	|                                                                                      |
	----------------------------------------------------------------------------------------

	Version history:
	Date        | Version   | Author       | Remark
	----------------------------------------------------------------------------------------
	28/10/2019  | 3.0       | L. Klar      | Initial version
	13/03/2020  | 3.1       | M. Kurpiers  | Adapting reviews
	16/01/2023  | 4.0       | S. Nikodem   | Release TIA 17 | DHL Munich 2023
	13/03/2023  | 4.1       | S. Nieswiec  | Updated for new Baseline
	*)

	REGION 1 – Update FIFO header status bits

	    // Mode 'S' - FIFO register status update.
	    "FC_Fifo"(ic_Mode := 'S',
	              qUDT_Status => #ss_Status.FIFOReceiveStatus,
	              qx_Error => #ss_Status.FIFOReceiveError,
	              qx_Warning => #ss_Status.FIFOReceiveWarning,
	              iqv_Data := #s_UDT_MessageArray,
	              iqUDT_FifoHeader := #iq_UDT_FifoHeader,
	              iqv_DataBuffer := #iqs_FifoData);

	END_REGION

	REGION 2 – Maximum number of message arrays elements

	    #si_MaximumMessageLength := "FC_GetNrOfArrayEl"(iv_Array := #s_UDT_MessageArray.Bytes);

	END_REGION

	REGION 3 – Receive enable

	    // Allow receiving if the connection is established and there are no FIFO errors.
	    #ss_TRCV.Enable :=
	    #ix_EnableReceive
	    AND NOT #ss_Status.FIFOReceiveError;

	    IF #si_BodyLength + #ii_HeaderLength > #si_MaximumMessageLength
	    THEN
	        #sx_STXFound := 0;
	        #sui_ReceivedMessageLength := 0;
	        #sx_ReceivedMessagePart := 0;
	        #sui_ReceivedMessagePartLength := 0;
	    END_IF;

	END_REGION

	REGION 4 – Receive data

	    // Data received in an ADHOC mode - data available immediately.
	    #s_FB_TRCV(EN_R := #ss_TRCV.Enable,
	               ID := #i_UDT_Connection.ID,
	               LEN := 0,
	               ADHOC := TRUE,
	               NDR => #ss_TRCV.NDR,
	               BUSY => #ss_TRCV.Busy,
	               ERROR => #ss_TRCV.Error,
	               STATUS => #ss_TRCV.Status,
	               RCVD_LEN => #ss_TRCV.ReceivedLength,
	               DATA := #ss_TRCV.Data);

	END_REGION

	REGION 5 – Received data handling

	    // Receiving data was successful.
	    IF #ss_TRCV.NDR
	        AND NOT #ss_TRCV.Busy
	        AND NOT #ss_TRCV.Error
	        AND #ss_TRCV.ReceivedLength > 0
	    THEN

	        REGION 5.1 – Initialization

	            #sui_ReceivedMessageLength := 0;
	            #sui_ReceivedMessagesOffset := 0;
	            #sui_NumberOfReceivedMessages := 0;

	        END_REGION

	        REGION 5.2 – Received part of the message

	            // Move part of the messages into a buffer if available.
	            IF #sx_ReceivedMessagePart
	            THEN
	                #s_UDT_MessageArray := #s_UDT_MessagePartArray;

	            END_IF;

	        END_REGION

	        REGION 5.3 – Message handling

	            FOR #ti_LC_MessageChars := 0 TO (UDINT_TO_INT(#ss_TRCV.ReceivedLength) - 1) DO
	                // Message length validation.
	                IF #sui_ReceivedMessageLength <= #si_MaximumMessageLength
	                THEN
	                    // First termination sign found.
	                    IF (#ss_TRCV.Data[#ti_LC_MessageChars] = #cb_STX)
	                        AND NOT #sx_STXFound
	                    THEN
	                        // Message didn't end.
	                        IF #ti_LC_MessageChars < UDINT_TO_INT(#ss_TRCV.ReceivedLength) - 1
	                        THEN
	                            // Second termination sign found.
	                            IF (#ss_TRCV.Data[#ti_LC_MessageChars + 1] = #cb_STX)
	                                OR #sx_STXFoundEnd
	                            THEN
	                                #sx_STXFound := TRUE;
	                                #sui_ReceivedMessagesOffset := #ti_LC_MessageChars;
	                                #sx_STXFoundEnd := FALSE;
	                            ELSE
	                                // Increment invalid meassage statistic.
	                                #iq_UDT_Statistics.InvalidMsg += 1;
	                            END_IF;
	                        ELSE
	                            #sui_ReceivedMessagesOffset := #ti_LC_MessageChars;
	                            #sx_STXFoundEnd := TRUE;
	                            #sui_ReceivedMessageLength := 1;
	                            #sui_ReceivedMessagePartLength := 1;
	                        END_IF;

	                    ELSIF #sx_STXFoundEnd
	                    THEN
	                        // Increment invalid meassage statistic and reset STX found signal.
	                        #iq_UDT_Statistics.InvalidMsg += 1;
	                        #sx_STXFoundEnd := FALSE;
	                    END_IF;

	                    // First STX is found.
	                    IF #sx_STXFound
	                    THEN
	                        // Increment received message length.
	                        #sui_ReceivedMessageLength += 1;

	                        // Take the second part of the body length from the message header.
	                        IF (#sui_ReceivedMessageLength + #sui_ReceivedMessagePartLength) = (#ii_BodyLengthPosition + 1)
	                        THEN
	                            #si_BodyLengthSecondPart := BYTE_TO_INT(#ss_TRCV.Data[#ti_LC_MessageChars]);
	                        END_IF;

	                        // Take the first part of the body length from the message header and add it to the first one.
	                        IF (#sui_ReceivedMessageLength + #sui_ReceivedMessagePartLength) = (#ii_BodyLengthPosition + 2)
	                        THEN
	                            #si_BodyLengthFirstPart := BYTE_TO_INT(#ss_TRCV.Data[#ti_LC_MessageChars]);
	                            #sw_BodyLength := INT_TO_WORD(IN := #si_BodyLengthFirstPart);
	                            #si_BodyLength := WORD_TO_INT(SHL(IN := #sw_BodyLength, N := 8)) + #si_BodyLengthSecondPart;
	                        END_IF;

	                        // When the whole message is received write it to the FIFO buffer.
	                        IF (#sui_ReceivedMessageLength + #sui_ReceivedMessagePartLength) = (#ii_HeaderLength + #si_BodyLength)
	                        THEN
	                            // Move received message to the message array.
	                            MOVE_BLK(IN := #ss_TRCV.Data[#sui_ReceivedMessagesOffset],
	                                     COUNT := #sui_ReceivedMessageLength,
	                                     OUT => #s_UDT_MessageArray.Bytes[#sui_ReceivedMessagePartLength]);  //#sui_ReceivedMessagePartLength

	                            // Clear not used message array characters.
	                            IF (#sui_ReceivedMessageLength + #sui_ReceivedMessagePartLength) < #si_MaximumMessageLength
	                            THEN
	                                FILL_BLK(IN := #cb_NULL,
	                                         COUNT := INT_TO_ULINT(#si_MaximumMessageLength) -
	                                         UDINT_TO_ULINT(#sui_ReceivedMessageLength) + #sui_ReceivedMessagePartLength,
	                                         OUT => #s_UDT_MessageArray.Bytes[#sui_ReceivedMessageLength + #sui_ReceivedMessagePartLength]);
	                            END_IF;

	                            // Mode 'W' - Write FIFO record.
	                            "FC_Fifo"(ic_Mode := 'W',
	                                      qUDT_Status => #ss_Status.FIFOReceiveStatus,
	                                      qx_Error => #ss_Status.FIFOReceiveError,
	                                      qx_Warning => #ss_Status.FIFOReceiveWarning,
	                                      iqv_Data := #s_UDT_MessageArray,
	                                      iqUDT_FifoHeader := #iq_UDT_FifoHeader,
	                                      iqv_DataBuffer := #iqs_FifoData);

	                            // Increment number of the received messages and initialize variables.
	                            #sui_NumberOfReceivedMessages += 1;
	                            #sui_ReceivedMessageLength := 0;
	                            #sui_ReceivedMessagePartLength := 0;
	                            #sx_ReceivedMessagePart := FALSE;
	                            #sx_STXFound := FALSE;
	                        END_IF;
	                    END_IF;
	                END_IF;
	            END_FOR;

	        END_REGION

	        REGION 5.4 – Part of the message preparation

	            // Only the part of the message is received.
	            IF (#sui_ReceivedMessageLength < #ii_HeaderLength + #si_BodyLength)
	                AND (#sx_STXFound OR #sx_STXFoundEnd)
	            THEN
	                // Clear not used message array characters.
	                FILL_BLK(IN := #cb_NULL,
	                         COUNT := INT_TO_ULINT(#si_MaximumMessageLength) -
	                         UDINT_TO_ULINT(#sui_ReceivedMessageLength),
	                         OUT => #s_UDT_MessagePartArray.Bytes[#sui_ReceivedMessageLength]);

	                // Move part of the message into a buffer.
	                MOVE_BLK(IN := #ss_TRCV.Data[#sui_ReceivedMessagesOffset],
	                         COUNT := #sui_ReceivedMessageLength,
	                         OUT => #s_UDT_MessagePartArray.Bytes[0]);

	                // Set the part of the message received bit and move length of the received message into the length of the part of the message variable.
	                #sx_ReceivedMessagePart := TRUE;
	                #sui_ReceivedMessagePartLength := #sui_ReceivedMessageLength;


	            END_IF;

	        END_REGION

	    END_IF;

	END_REGION

	REGION 6 – Status

	    REGION 6.1 - Block status

	        // Receive error.
	        #ss_Status.ReceiveError := #ss_TRCV.Error;

	        // Parametrization collective error output.
	        #qx_Error :=
	        #ss_Status.FIFOReceiveError
	        OR #ss_Status.ReceiveError;

	        // Parametrization collective warning output.
	        #qx_Warning := #ss_Status.FIFOReceiveWarning;

	    END_REGION

	    REGION 6.2 - Error code preparation

	        IF #ss_TRCV.#Status > 16#8000
	            OR #ss_TRCV.#Status = 16#0
	        THEN
	            #ss_Status.ErrorCode.TRCV := #ss_TRCV.#Status;
	        END_IF;

	    END_REGION
	END_REGION
END_FUNCTION_BLOCK

FUNCTION_BLOCK "FB_MFC_Visu_ArmDiverter_Status"
{ S7_Optimized_Access := 'TRUE' }
VERSION : 0.1
// ATTRIBUTES
// AUTO_NUMBER = True
// BLOCK_NUMBER = 135
// END_ATTRIBUTES
   VAR_INPUT
      i_UDT_ArmDiverterStatus { ExternalAccessible := 'False'; ExternalVisible := 'False'; ExternalWritable := 'False'} : "UDT_ArmDiverterStatus";   // ArmDiverter status structure
      i_UDT_EquipmentNumber { ExternalAccessible := 'False'; ExternalVisible := 'False'; ExternalWritable := 'False'} : "UDT_EquipmentNumber";   // Item number
      ix_SendAllErrorsState { ExternalAccessible := 'False'; ExternalVisible := 'False'; ExternalWritable := 'False'} : Bool;   // True - update all the messages
      ix_MFCConnected { ExternalAccessible := 'False'; ExternalVisible := 'False'; ExternalWritable := 'False'} : Bool;   // True - A connection to the MFC has been established
      ix_CollectiveReset { ExternalAccessible := 'False'; ExternalVisible := 'False'; ExternalWritable := 'False'} : Bool;   // True - Collective reset command of all system controls
   END_VAR

   VAR_OUTPUT
      qx_Error { ExternalAccessible := 'False'; ExternalVisible := 'False'; ExternalWritable := 'False'} : Bool;   // Block error
      qx_Warning { ExternalAccessible := 'False'; ExternalVisible := 'False'; ExternalWritable := 'False'} : Bool;   // Block warning
   END_VAR

   VAR_IN_OUT
      iq_UDT_FifoHeader : "UDT_FifoHeader";   // FIFO header
      iqs_FifoData : Array[*] of "UDT_MessageV2";   // FIFO data buffer
      iqdi_MessageSequenceNumber { ExternalAccessible := 'False'; ExternalVisible := 'False'; ExternalWritable := 'False'} : DInt;   // Message number
   END_VAR

   VAR
      s_FB_ItemStatus { ExternalAccessible := 'False'; ExternalVisible := 'False'; ExternalWritable := 'False'; S7_SetPoint := 'False'} : "FB_ItemStatus";   // Item status block's instance
      s_FB_ItemError { ExternalAccessible := 'False'; ExternalVisible := 'False'; ExternalWritable := 'False'; S7_SetPoint := 'False'} : "FB_ItemError";   // Item error block's instance
      ss_FIFOStatus { ExternalAccessible := 'False'; ExternalVisible := 'False'; ExternalWritable := 'False'; S7_SetPoint := 'False'} : "UDT_FifoStatus";   // Status structure
      s_UDT_Message { ExternalAccessible := 'False'; ExternalVisible := 'False'; ExternalWritable := 'False'; S7_SetPoint := 'False'} : "UDT_Message";   // Message
      s_UDT_ItemStatus { ExternalAccessible := 'False'; ExternalVisible := 'False'; ExternalWritable := 'False'; S7_SetPoint := 'False'} : "UDT_ItemStatus";   // Item status message body structure
      s_UDT_ArmDiverterOldStatus { ExternalAccessible := 'False'; ExternalVisible := 'False'; ExternalWritable := 'False'; S7_SetPoint := 'False'} : "UDT_ArmDiverterStatus";   // ArmDiverter  old status structure
      s_UDT_ItemError { ExternalAccessible := 'False'; ExternalVisible := 'False'; ExternalWritable := 'False'; S7_SetPoint := 'False'} : "UDT_ItemError";   // Item error message body structure
      s_R_TRIG_Connection {InstructionName := 'R_TRIG'; LibVersion := '1.0'; ExternalAccessible := 'False'; ExternalVisible := 'False'; ExternalWritable := 'False'; S7_SetPoint := 'False'} : R_TRIG;   // Rising edge trigger connection reastablished
      s_F_TRIG_SendAllErrors {InstructionName := 'F_TRIG'; LibVersion := '1.0'; ExternalAccessible := 'False'; ExternalVisible := 'False'; ExternalWritable := 'False'; S7_SetPoint := 'False'} : F_TRIG;   // Falling edge trigger from signal send all errors
      sdi_Code { ExternalAccessible := 'False'; ExternalVisible := 'False'; ExternalWritable := 'False'} : DInt;   // Error code
      si_ItemStatus { ExternalAccessible := 'False'; ExternalVisible := 'False'; ExternalWritable := 'False'} : Int;   // Item status
      ii_ErrorNumber { ExternalAccessible := 'False'; ExternalVisible := 'False'; ExternalWritable := 'False'} : Int;   // Counter Error Number
      si_State { ExternalAccessible := 'False'; ExternalVisible := 'False'; ExternalWritable := 'False'} : Int;   // Error state
      sx_ItemErrorMessageReq { ExternalAccessible := 'False'; ExternalVisible := 'False'; ExternalWritable := 'False'} : Bool;   // Item error message required
      sx_ItemStatusMessageReq { ExternalAccessible := 'False'; ExternalVisible := 'False'; ExternalWritable := 'False'} : Bool;   // Item status message required
      sx_SendAllProcedure { ExternalAccessible := 'False'; ExternalVisible := 'False'; ExternalWritable := 'False'} : Bool;   // Send all procedure
      sx_FIFOError { ExternalAccessible := 'False'; ExternalVisible := 'False'; ExternalWritable := 'False'} : Bool;   // FIFO error
      sx_FIFOWarning { ExternalAccessible := 'False'; ExternalVisible := 'False'; ExternalWritable := 'False'} : Bool;   // FIFO warning
      sx_ItemErrorBlockError { ExternalAccessible := 'False'; ExternalVisible := 'False'; ExternalWritable := 'False'} : Bool;   // Item error block error
      sx_ItemErrorBlockWarning { ExternalAccessible := 'False'; ExternalVisible := 'False'; ExternalWritable := 'False'} : Bool;   // Item error block warning
      sx_ItemStatusBlockError { ExternalAccessible := 'False'; ExternalVisible := 'False'; ExternalWritable := 'False'} : Bool;   // Item status block error
      sx_ItemStatusBlockWarning { ExternalAccessible := 'False'; ExternalVisible := 'False'; ExternalWritable := 'False'} : Bool;   // Item status block warning
   END_VAR


BEGIN
	(*
	----------------------------------------------------------------------------------------
	|                                                                                      |
	|  Copyright  2023             FORTNA Europe BV                                        |
	|  All Rights Reserved         Netherlands                                             |
	|                                                                                      |
	----------------------------------------------------------------------------------------
	Version history:
	Date        | Version   | Author       | Remark
	----------------------------------------------------------------------------------------
	21/03/2023  | 1.0       | M. Diebel   | Release TIA 17 | DHL Munich 2023
	04/03/2024  | 1.1       | M. Diebel   | Release TIA 17 | incremant #ii_ErrorNumber for reference error
	13/03/2024  | 1.2       | S. Nieswiec | Updated for new Baseline
	*)


	REGION 1 - Initialize message required signals

	    #sx_ItemErrorMessageReq := FALSE;
	    #sx_ItemStatusMessageReq := FALSE;

	    // On connection reestablish send last remembered status and error state ( status only when it's diffrent then 0 )
	    #s_R_TRIG_Connection(CLK := #ix_MFCConnected);

	    IF #s_R_TRIG_Connection.Q AND #si_ItemStatus <> 0
	    THEN
	        #sx_ItemStatusMessageReq := TRUE;
	    END_IF;

	    IF #s_R_TRIG_Connection.Q
	    THEN
	        #sx_ItemErrorMessageReq := TRUE;
	    END_IF;

	    // Prepare trigger on the collective reset signal.
	    #s_F_TRIG_SendAllErrors(CLK := #ix_SendAllErrorsState);

	    // When collective reset will go down, start send every equipment errors.
	    IF #s_F_TRIG_SendAllErrors.Q AND NOT #sx_SendAllProcedure
	    THEN
	        #ii_ErrorNumber := 0;
	        #sx_SendAllProcedure := TRUE;
	    END_IF;

	END_REGION

	REGION 2 - FIFO header status update

	    // Mode 'S' - FIFO register status update.
	    "FC_Fifo"(ic_Mode := 'S',
	              qUDT_Status => #ss_FIFOStatus,
	              qx_Error => #sx_FIFOError,
	              qx_Warning => #sx_FIFOWarning,
	              iqv_Data := #s_UDT_Message,
	              iqUDT_FifoHeader := #iq_UDT_FifoHeader,
	              iqv_DataBuffer := #iqs_FifoData);

	END_REGION

	REGION 3 - Prepare message data

	    // When there is no reset errors command, update status and errors.
	    IF NOT #ix_CollectiveReset
	        AND NOT #ss_FIFOStatus.FifoPreFull
	    THEN
	        // Status
	        IF (#i_UDT_ArmDiverterStatus.Status <> #s_UDT_ArmDiverterOldStatus.Status OR (#sx_SendAllProcedure AND #ii_ErrorNumber = 0))
	        THEN
	            #sx_ItemStatusMessageReq := TRUE;
	            #si_ItemStatus := #i_UDT_ArmDiverterStatus.Status;
	            #s_UDT_ArmDiverterOldStatus.Status := #i_UDT_ArmDiverterStatus.Status;
	        END_IF;


